(* Logix 5000 project; controller ACMI_PLC vendor 1 type 14 code 101 rev 19.11; software revision 19.01 *)
// Safety Rated PLC

TASK MainTask (periodic, rate 100 ms, priority 10, watchdog 2000 ms) : MainProgram
TASK SafetyTask (periodic, rate 20 ms, priority 2, watchdog 20 ms) : Main_Loop

MODULES
   Local : vendor 1 type 14 code 101 (1768Ctrl3Slot 0, Compact 0, rev 19.11)
      Temps : 1769-IR6 (Compact 1, rev 1.1, Input RPI 80 ms)
      SafetyEthernet : 1768-ENBT (1768 1, Ethernet 192.168.1.8, rev 4.4)
         PointIONet : 1734-AENT (Ethernet 192.168.1.9, rev 4.3, Output RPI 20 ms)
             : vendor 1 type 35 code 15 (PointIO 1, rev 2.1, Output RPI 20 ms, Input RPI 10 ms)
             : vendor 1 type 35 code 15 (PointIO 5, rev 2.1, Output RPI 20 ms, Input RPI 10 ms)
             : vendor 1 type 35 code 16 (PointIO 6, rev 2.1, Input RPI 10 ms, Output RPI 20 ms)
             : vendor 1 type 35 code 15 (PointIO 2, rev 2.1, Input RPI 10 ms, Output RPI 20 ms)
             : vendor 1 type 35 code 15 (PointIO 7, rev 2.1, Input RPI 10 ms, Output RPI 20 ms)
             : vendor 1 type 35 code 15 (PointIO 3, rev 2.1, Output RPI 20 ms, Input RPI 10 ms)
             : vendor 1 type 35 code 15 (PointIO 4, rev 2.1, Output RPI 20 ms, Input RPI 10 ms)
      PGRM : 1768-ENBT (1768 2, Ethernet 10.0.128.19, rev 4.1)
END_MODULES

TYPE BitStat :
STRUCT
   Hist : BOOL[4096];
   Top : INT;
   Sum : INT;
   Fault : BOOL;
END_STRUCT
END_TYPE

TYPE EVENT :
STRUCT
   TIME : TIME;
   EVENT : STRING;
END_STRUCT
END_TYPE

TYPE TIME :
STRUCT
   YEAR : DINT;
   MONTH : DINT;
   DAY : DINT;
   HOUR : DINT;
   MINUTE : DINT;
   SECOND : DINT;
   MICROSECOND : DINT;
END_STRUCT
END_TYPE

VAR_GLOBAL   (* controller tags *)
   A : DINT := 2047; {access Read Only}
   Abits : INT;
   ACMI_ADC_BITS : INT[2]; {access Read Only}
   ACMI_BEAM_DATA : REAL[7] := ([0] := 19.653, [1] := 16.0, [2] := -0.15, [5] := 82.0, [6] := 0.03); {access Read Only}
   ACMI_BEAM_Q : REAL := 19.653; {access Read Only}
   ACMI_BR_ACC : REAL; {access Read Only}
   ACMI_BR_CNT : DINT := 3278; {access Read Only}
   ACMI_BR_LIM : REAL := 82.0; {access Read Only}
   ACMI_CERTIFY : SINT; {access Read Only}
   ACMI_FAULT_CODE : DINT := 2097063; {access Read Only}
   ACMI_SHUTTER : BOOL; {access Read Only}
   ACMI_SR_LIM : REAL := 0.03; {access Read Only}
   ACMI_ST1_QAB : REAL := 19.021; {access Read Only}
   ACMI_ST1_QAB_AVG : REAL := 18.336615; {access Read Only}
   ACMI_ST1_QAB_HIST : DINT[31] := ([30] := 200); {access Read Only}
   ACMI_ST1_QAB_MAX : REAL := 19.713; {access Read Only}
   ACMI_ST1_QAB_MIN : REAL := -17.556; {access Read Only}
   ACMI_ST1_QAB_STD : REAL := 3362.0618; {access Read Only}
   ACMI_ST1_QBA : REAL := 19.152; {access Read Only}
   ACMI_ST1_QBA_AVG : REAL := 18.44839; {access Read Only}
   ACMI_ST1_QBA_HIST : DINT[31] := ([30] := 200); {access Read Only}
   ACMI_ST1_QBA_MAX : REAL := 19.713; {access Read Only}
   ACMI_ST1_QBA_MIN : REAL := -17.613; {access Read Only}
   ACMI_ST1_QBA_STD : REAL := 3396.1123; {access Read Only}
   ACMI_ST1_RST : SINT; {access Read Only}
   ACMI_ST2_QAB : REAL := 19.062; {access Read Only}
   ACMI_ST2_QAB_AVG : REAL := 18.345718; {access Read Only}
   ACMI_ST2_QAB_HIST : DINT[31] := ([30] := 200); {access Read Only}
   ACMI_ST2_QAB_MAX : REAL := 19.713; {access Read Only}
   ACMI_ST2_QAB_MIN : REAL := -17.572; {access Read Only}
   ACMI_ST2_QAB_STD : REAL := 3360.6584; {access Read Only}
   ACMI_ST2_QBA : REAL := 19.132; {access Read Only}
   ACMI_ST2_QBA_AVG : REAL := 18.451597; {access Read Only}
   ACMI_ST2_QBA_HIST : DINT[31] := ([30] := 200); {access Read Only}
   ACMI_ST2_QBA_MAX : REAL := 19.713; {access Read Only}
   ACMI_ST2_QBA_MIN : REAL := -17.638; {access Read Only}
   ACMI_ST2_QBA_STD : REAL := 3401.8562; {access Read Only}
   ACMI_ST2_RST : SINT; {access None}
   ACMI_ST_DATA : REAL[24] := ([0] := 19.021, [1] := 18.336615, [2] := 19.713, [3] := -17.556, [4] := 3362.0618, [5] := 19.152, [6] := 18.44839, [7] := 19.713, [8] := -17.613, [9] := 3396.1123, [10] := 0.75, [11] := 0.35, [12] := 19.062, [13] := 18.345718, [14] := 19.713, [15] := -17.572, [16] := 3360.6584, [17] := 19.132, [18] := 18.451597, [19] := 19.713, [20] := -17.638, [21] := 3401.8562, [22] := 16.4, [23] := 15.4); {access Read Only}
   ACMI_STAT_CODE : SINT; {access Read Only}
   ACMI_Stat_Size : INT := 200; {access Read Only}
   ACMI_TEMPS : INT[6] := ([0] := 210, [1] := 394, [2] := 256, [3] := 213, [4] := 172, [5] := 214); {access Read Only}
   ACMI_TIMING : SINT; {access Read Only}
   ACMI_TO_ACC : REAL; {access Read Only}
   ACMI_TO_CNT : DINT := 39; {access Read Only}
   ADCA : DINT := 2047; {access Read Only}
   ADCB : DINT := 58; {access Read Only}
   B : DINT := 58; {access Read Only}
   Bbits : INT;
   Beam_MaxQ : DINT := 16000; {constant, access Read Only}
   Beam_MinQ : DINT := -150; {constant, access Read Only}
   Beam_Q : DINT := 19653; {access Read Only}
   BR_Stack : DINT[7200]; {access Read Only}
   BR_Stack_MAX : DINT := 82000000; {constant, access Read Only}
   BR_Stack_Sum : DINT; {access Read Only}
   BR_Stack_Top : DINT := 923; {access Read Only}
   BSSS_CLOSED : ALIAS FOR PointIONet:7:I.Pt00Data;
   BYPASS_KEY : ALIAS FOR PointIONet:5:I.Pt07Data;
   FAULT_BEAM_BL : BOOL := 1; {access Read Only}
   FAULT_BEAM_HI : BOOL := 1; {access Read Only}
   FAULT_BEAM_LO : BOOL := 1;
   FAULT_BR_ACC : BOOL; {access Read Only}
   FAULT_CODE : DINT := 2097063;
   FAULT_QOW1 : BOOL := 1; {access Read Only}
   FAULT_QOW2 : BOOL; {access Read Only}
   FAULT_ST1_AB_HI : BOOL := 1; {access Read Only}
   FAULT_ST1_AB_LO : BOOL := 1; {access Read Only}
   FAULT_ST1_BA_HI : BOOL := 1; {access Read Only}
   FAULT_ST1_BA_LO : BOOL := 1; {access Read Only}
   FAULT_ST1_BLA : BOOL := 1; {access Read Only}
   FAULT_ST1_BLB : BOOL := 1; {access Read Only}
   FAULT_ST1_QAT : BOOL := 1; {access Read Only}
   FAULT_ST2_AB_HI : BOOL := 1; {access Read Only}
   FAULT_ST2_AB_LO : BOOL := 1; {access Read Only}
   FAULT_ST2_BA_HI : BOOL := 1; {access Read Only}
   FAULT_ST2_BA_LO : BOOL := 1; {access Read Only}
   FAULT_ST2_BLA : BOOL := 1; {access Read Only}
   FAULT_ST2_BLB : BOOL := 1; {access Read Only}
   FAULT_ST2_QAT : BOOL := 1; {access Read Only}
   FAULT_TO_ACC : BOOL; {access Read Only}
   FAULT_TWB : BOOL; {access Read Only}
   FAULT_WDT : BOOL; {access Read Only}
   HMI_BEAM_Q : REAL := 19.653; {access Read Only}
   HMI_Suppress : BOOL;
   Initialize : BOOL := 1; {access Read Only}
   LBSS_CLOSED : ALIAS FOR PointIONet:7:I.Pt01Data;
   PPS_RESET : ALIAS FOR PointIONet:7:I.Pt02Data;
   Q1AB : DINT;
   Relay_Error : BOOL; {access Read Only}
   RESET_ALL : ALIAS FOR PointIONet:5:I.Pt00Data;
   RESET_FAULT : ALIAS FOR PointIONet:5:I.Pt01Data;
   ST1_MaxQ : DINT := 750; {constant}
   ST1_MinQ : DINT := 350; {constant}
   ST1_QAB : DINT := 19021;
   ST1_QBA : DINT := 19152;
   ST1AB_Size : INT := 200;
   ST1BA_Size : INT := 200;
   ST2_MaxQ : DINT := 16400; {constant}
   ST2_MinQ : DINT := 15400; {constant}
   ST2_QAB : DINT := 19062;
   ST2_QBA : DINT := 19132;
   ST2AB_Size : INT := 200;
   ST2BA_Size : INT := 200;
   ST_HI_FAULT : BOOL := 1; {access Read Only}
   ST_LO_FAULT : BOOL; {access Read Only}
   ST_Size : BOOL := 1;
   ST_Type : BOOL;
   Stack_Size : DINT := 7067; {constant, access Read Only}
   TO_Cntr : COUNTER;
   TO_DISABLED : ALIAS FOR PointIONet:7:I.Pt03Data;
   TO_Stack : DINT[120]; {access Read Only}
   TO_Stack_MAX : DINT := 30000; {constant, access Read Only}
   TO_Stack_Size : DINT := 118; {constant, access Read Only}
   TO_Stack_Sum : DINT; {access Read Only}
   TO_Stack_Top : DINT := 47;
   TO_Status_Error : BOOL;
   Update_ST1_QAB : BOOL;
   Update_ST1_QBA : BOOL := 1;
   Update_ST2_QAB : BOOL := 1;
   Update_ST2_QBA : BOOL;
   Zero : DINT[7200]; {constant}
END_VAR

PROGRAM Event_Log   (* main routine Event_Log *)
VAR
   action_1 : BOOL; {access Read Only}
   action_10 : BOOL := 1; {access Read Only}
   action_11 : BOOL := 1;
   action_12 : BOOL;
   action_2 : BOOL := 1; {access Read Only}
   action_3 : BOOL; {access Read Only}
   action_4 : BOOL := 1; {access Read Only}
   action_5 : BOOL := 1; {access Read Only}
   action_6 : BOOL; {access Read Only}
   action_7 : BOOL := 1; {access Read Only}
   action_8 : BOOL; {access Read Only}
   action_9 : BOOL := 1; {access Read Only}
   Clear_Elog : BOOL := 1;
   Clock : TIME := (YEAR := 2025, MONTH := 4, DAY := 25, HOUR := 11, MINUTE := 37, SECOND := 34, MICROSECOND := 91157); {access Read Only}
   colon : STRING := ':'; {constant, access Read Only}
   Ehome : BOOL;
   Ehomeons : BOOL;
   Eindx : DINT;
   ELog : EVENT[1000] := ([0].TIME.YEAR := 2016, [0].TIME.MONTH := 6, [0].TIME.DAY := 14, [0].TIME.HOUR := 8, [0].TIME.MINUTE := 54, [0].TIME.SECOND := 13, [0].TIME.MICROSECOND := 99494, [0].EVENT := '2016/06/14   08:54:13   USER : RESET FAULT BUTTON PRESSED', [1].TIME.YEAR := 2016, [1].TIME.MONTH := 6, [1].TIME.DAY := 14, [1].TIME.HOUR := 15, [1].TIME.MINUTE := 7, [1].TIME.SECOND := 39, [1].TIME.MICROSECOND := 999465, [1].EVENT := '2016/06/14   15:07:39   FAULT : QOW1 : Charge Outside Window Detected', [2].TIME.YEAR := 2016, [2].TIME.MONTH := 6, [2].TIME.DAY := 14, [2].TIME.HOUR := 18, [2].TIME.MINUTE := 16, [2].TIME.SECOND := 9, [2].TIME.MICROSECOND := 400030, [2].EVENT := '2016/06/14   18:16:09   USER : PPS RESET FAULT BUTTON PRESSED', [3].TIME.YEAR := 2016, [3].TIME.MONTH := 6, [3].TIME.DAY := 14, [3].TIME.HOUR := 18, [3].TIME.MINUTE := 18, [3].TIME.SECOND := 25, [3].TIME.MICROSECOND := 799513, [3].EVENT := '2016/06/14   18:18:25   USER : PPS RESET FAULT BUTTON PRESSED', [4].TIME.YEAR := 2016, [4].TIME.MONTH := 6, [4].TIME.DAY := 14, [4].TIME.HOUR := 18, [4].TIME.MINUTE := 25, [4].TIME.SECOND := 9, [4].TIME.MICROSECOND := 99507, [4].EVENT := '2016/06/14   18:25:09   USER : PPS RESET FAULT BUTTON PRESSED', [5].TIME.YEAR := 2016, [5].TIME.MONTH := 6, [5].TIME.DAY := 14, [5].TIME.HOUR := 18, [5].TIME.MINUTE := 32, [5].TIME.SECOND := 13, [5].TIME.MICROSECOND := 899509, [5].EVENT := '2016/06/14   18:32:13   USER : PPS RESET FAULT BUTTON PRESSED', [6].TIME.YEAR := 2016, [6].TIME.MONTH := 6, [6].TIME.DAY := 14, [6].TIME.HOUR := 18, [6].TIME.MINUTE := 32, [6].TIME.SECOND := 14, [6].TIME.MICROSECOND := 399506, [6].EVENT := '2016/06/14   18:32:14   USER : PPS RESET FAULT BUTTON PRESSED', [7].TIME.YEAR := 2016, [7].TIME.MONTH := 6, [7].TIME.DAY := 14, [7].TIME.HOUR := 18,
        [7].TIME.MINUTE := 33, [7].TIME.SECOND := 34, [7].TIME.MICROSECOND := 499505, [7].EVENT := '2016/06/14   18:33:34   USER : PPS RESET FAULT BUTTON PRESSED', [8].TIME.YEAR := 2016, [8].TIME.MONTH := 6, [8].TIME.DAY := 14, [8].TIME.HOUR := 19, [8].TIME.MINUTE := 20, [8].TIME.SECOND := 22, [8].TIME.MICROSECOND := 599510, [8].EVENT := '2016/06/14   19:20:22   USER : PPS RESET FAULT BUTTON PRESSED', [9].TIME.YEAR := 2016, [9].TIME.MONTH := 6, [9].TIME.DAY := 14, [9].TIME.HOUR := 19, [9].TIME.MINUTE := 30, [9].TIME.SECOND := 2, [9].TIME.MICROSECOND := 699510, [9].EVENT := '2016/06/14   19:30:02   USER : PPS RESET FAULT BUTTON PRESSED', [10].TIME.YEAR := 2016, [10].TIME.MONTH := 6, [10].TIME.DAY := 14, [10].TIME.HOUR := 19, [10].TIME.MINUTE := 49, [10].TIME.SECOND := 34, [10].TIME.MICROSECOND := 999476, [10].EVENT := '2016/06/14   19:49:34   FAULT : QOW1 : Charge Outside Window Detected', [11].TIME.YEAR := 2016, [11].TIME.MONTH := 6, [11].TIME.DAY := 14, [11].TIME.HOUR := 19, [11].TIME.MINUTE := 50, [11].TIME.SECOND := 16, [11].TIME.MICROSECOND := 499512, [11].EVENT := '2016/06/14   19:50:16   USER : PPS RESET FAULT BUTTON PRESSED', [12].TIME.YEAR := 2016, [12].TIME.MONTH := 6, [12].TIME.DAY := 14, [12].TIME.HOUR := 19, [12].TIME.MINUTE := 50, [12].TIME.SECOND := 17, [12].TIME.MICROSECOND := 999514, [12].EVENT := '2016/06/14   19:50:17   USER : PPS RESET FAULT BUTTON PRESSED', [13].TIME.YEAR := 2016, [13].TIME.MONTH := 6, [13].TIME.DAY := 14, [13].TIME.HOUR := 19, [13].TIME.MINUTE := 58, [13].TIME.SECOND := 36, [13].TIME.MICROSECOND := 900080, [13].EVENT := '2016/06/14   19:58:36   USER : PPS RESET FAULT BUTTON PRESSED', [14].TIME.YEAR := 2016, [14].TIME.MONTH := 6, [14].TIME.DAY := 14, [14].TIME.HOUR := 21, [14].TIME.MINUTE := 23, [14].TIME.SECOND := 39, [14].TIME.MICROSECOND := 799512, [14].EVENT := '2016/06/14   21:23:39   USER : PPS RESET FAULT BUTTON PRESSED',
        [15].TIME.YEAR := 2016, [15].TIME.MONTH := 6, [15].TIME.DAY := 14, [15].TIME.HOUR := 22, [15].TIME.MINUTE := 11, [15].TIME.SECOND := 59, [15].TIME.MICROSECOND := 800029, [15].EVENT := '2016/06/14   22:11:59   USER : PPS RESET FAULT BUTTON PRESSED', [16].TIME.YEAR := 2016, [16].TIME.MONTH := 6, [16].TIME.DAY := 14, [16].TIME.HOUR := 23, [16].TIME.MINUTE := 1, [16].TIME.SECOND := 6, [16].TIME.MICROSECOND := 699515, [16].EVENT := '2016/06/14   23:01:06   USER : PPS RESET FAULT BUTTON PRESSED', [17].TIME.YEAR := 2016, [17].TIME.MONTH := 6, [17].TIME.DAY := 15, [17].TIME.MINUTE := 55, [17].TIME.SECOND := 57, [17].TIME.MICROSECOND := 899506, [17].EVENT := '2016/06/15   00:55:57   USER : PPS RESET FAULT BUTTON PRESSED', [18].TIME.YEAR := 2016, [18].TIME.MONTH := 6, [18].TIME.DAY := 15, [18].TIME.HOUR := 1, [18].TIME.MINUTE := 43, [18].TIME.SECOND := 11, [18].TIME.MICROSECOND := 799939, [18].EVENT := '2016/06/15   01:43:11   USER : PPS RESET FAULT BUTTON PRESSED', [19].TIME.YEAR := 2016, [19].TIME.MONTH := 6, [19].TIME.DAY := 15, [19].TIME.HOUR := 2, [19].TIME.MINUTE := 28, [19].TIME.SECOND := 20, [19].TIME.MICROSECOND := 599507, [19].EVENT := '2016/06/15   02:28:20   USER : PPS RESET FAULT BUTTON PRESSED', [20].TIME.YEAR := 2016, [20].TIME.MONTH := 6, [20].TIME.DAY := 15, [20].TIME.HOUR := 3, [20].TIME.MINUTE := 26, [20].TIME.SECOND := 38, [20].TIME.MICROSECOND := 999502, [20].EVENT := '2016/06/15   03:26:38   USER : PPS RESET FAULT BUTTON PRESSED', [21].TIME.YEAR := 2016, [21].TIME.MONTH := 6, [21].TIME.DAY := 15, [21].TIME.HOUR := 4, [21].TIME.MINUTE := 11, [21].TIME.SECOND := 32, [21].TIME.MICROSECOND := 999506, [21].EVENT := '2016/06/15   04:11:32   USER : PPS RESET FAULT BUTTON PRESSED', [22].TIME.YEAR := 2016, [22].TIME.MONTH := 6, [22].TIME.DAY := 15, [22].TIME.HOUR := 4, [22].TIME.MINUTE := 50,
        [22].TIME.SECOND := 6, [22].TIME.MICROSECOND := 899508, [22].EVENT := '2016/06/15   04:50:06   USER : PPS RESET FAULT BUTTON PRESSED', [23].TIME.YEAR := 2016, [23].TIME.MONTH := 6, [23].TIME.DAY := 15, [23].TIME.HOUR := 5, [23].TIME.MINUTE := 8, [23].TIME.SECOND := 40, [23].TIME.MICROSECOND := 199505, [23].EVENT := '2016/06/15   05:08:40   USER : PPS RESET FAULT BUTTON PRESSED', [24].TIME.YEAR := 2016, [24].TIME.MONTH := 6, [24].TIME.DAY := 15, [24].TIME.HOUR := 5, [24].TIME.MINUTE := 36, [24].TIME.SECOND := 52, [24].TIME.MICROSECOND := 99507, [24].EVENT := '2016/06/15   05:36:52   USER : PPS RESET FAULT BUTTON PRESSED', [25].TIME.YEAR := 2016, [25].TIME.MONTH := 6, [25].TIME.DAY := 15, [25].TIME.HOUR := 7, [25].TIME.MINUTE := 29, [25].TIME.SECOND := 5, [25].TIME.MICROSECOND := 499507, [25].EVENT := '2016/06/15   07:29:05   USER : PPS RESET FAULT BUTTON PRESSED', [26].TIME.YEAR := 2016, [26].TIME.MONTH := 6, [26].TIME.DAY := 15, [26].TIME.HOUR := 9, [26].TIME.MINUTE := 57, [26].TIME.SECOND := 54, [26].TIME.MICROSECOND := 799464, [26].EVENT := '2016/06/15   09:57:54   FAULT : QOW1 : Charge Outside Window Detected', [27].TIME.YEAR := 2016, [27].TIME.MONTH := 6, [27].TIME.DAY := 15, [27].TIME.HOUR := 12, [27].TIME.MINUTE := 48, [27].TIME.SECOND := 48, [27].TIME.MICROSECOND := 999725, [27].EVENT := '2016/06/15   12:48:48   USER : PPS RESET FAULT BUTTON PRESSED', [28].TIME.YEAR := 2016, [28].TIME.MONTH := 6, [28].TIME.DAY := 15, [28].TIME.HOUR := 16, [28].TIME.MINUTE := 54, [28].TIME.SECOND := 28, [28].TIME.MICROSECOND := 299521, [28].EVENT := '2016/06/15   16:54:28   USER : PPS RESET FAULT BUTTON PRESSED', [29].TIME.YEAR := 2016, [29].TIME.MONTH := 6, [29].TIME.DAY := 15, [29].TIME.HOUR := 17, [29].TIME.MINUTE := 29, [29].TIME.SECOND := 30, [29].TIME.MICROSECOND := 299467, [29].EVENT := '2016/06/15   17:29:30   FAULT : QOW1 : Charge Outside Window Detected', [30].TIME.YEAR := 2016,
        [30].TIME.MONTH := 6, [30].TIME.DAY := 15, [30].TIME.HOUR := 17, [30].TIME.MINUTE := 30, [30].TIME.MICROSECOND := 600025, [30].EVENT := '2016/06/15   17:30:00   USER : PPS RESET FAULT BUTTON PRESSED', [31].TIME.YEAR := 2016, [31].TIME.MONTH := 6, [31].TIME.DAY := 15, [31].TIME.HOUR := 17, [31].TIME.MINUTE := 30, [31].TIME.SECOND := 48, [31].TIME.MICROSECOND := 99559, [31].EVENT := '2016/06/15   17:30:48   USER : PPS RESET FAULT BUTTON PRESSED', [32].TIME.YEAR := 2016, [32].TIME.MONTH := 6, [32].TIME.DAY := 15, [32].TIME.HOUR := 17, [32].TIME.MINUTE := 31, [32].TIME.SECOND := 16, [32].TIME.MICROSECOND := 999943, [32].EVENT := '2016/06/15   17:31:16   USER : PPS RESET FAULT BUTTON PRESSED', [33].TIME.YEAR := 2016, [33].TIME.MONTH := 6, [33].TIME.DAY := 15, [33].TIME.HOUR := 17, [33].TIME.MINUTE := 31, [33].TIME.SECOND := 20, [33].TIME.MICROSECOND := 699565, [33].EVENT := '2016/06/15   17:31:20   USER : PPS RESET FAULT BUTTON PRESSED', [34].TIME.YEAR := 2016, [34].TIME.MONTH := 6, [34].TIME.DAY := 15, [34].TIME.HOUR := 17, [34].TIME.MINUTE := 33, [34].TIME.SECOND := 7, [34].TIME.MICROSECOND := 599508, [34].EVENT := '2016/06/15   17:33:07   USER : PPS RESET FAULT BUTTON PRESSED', [35].TIME.YEAR := 2016, [35].TIME.MONTH := 6, [35].TIME.DAY := 15, [35].TIME.HOUR := 17, [35].TIME.MINUTE := 37, [35].TIME.SECOND := 31, [35].TIME.MICROSECOND := 400126, [35].EVENT := '2016/06/15   17:37:31   USER : PPS RESET FAULT BUTTON PRESSED', [36].TIME.YEAR := 2016, [36].TIME.MONTH := 6, [36].TIME.DAY := 15, [36].TIME.HOUR := 17, [36].TIME.MINUTE := 37, [36].TIME.SECOND := 35, [36].TIME.MICROSECOND := 18, [36].EVENT := '2016/06/15   17:37:35   USER : PPS RESET FAULT BUTTON PRESSED', [37].TIME.YEAR := 2016, [37].TIME.MONTH := 6, [37].TIME.DAY := 15, [37].TIME.HOUR := 22, [37].TIME.MINUTE := 8, [37].TIME.SECOND := 46,
        [37].TIME.MICROSECOND := 799505, [37].EVENT := '2016/06/15   22:08:46   USER : PPS RESET FAULT BUTTON PRESSED', [38].TIME.YEAR := 2016, [38].TIME.MONTH := 6, [38].TIME.DAY := 15, [38].TIME.HOUR := 22, [38].TIME.MINUTE := 26, [38].TIME.SECOND := 18, [38].TIME.MICROSECOND := 799507, [38].EVENT := '2016/06/15   22:26:18   USER : PPS RESET FAULT BUTTON PRESSED', [39].TIME.YEAR := 2016, [39].TIME.MONTH := 6, [39].TIME.DAY := 15, [39].TIME.HOUR := 22, [39].TIME.MINUTE := 26, [39].TIME.SECOND := 19, [39].TIME.MICROSECOND := 999507, [39].EVENT := '2016/06/15   22:26:19   USER : PPS RESET FAULT BUTTON PRESSED', [40].TIME.YEAR := 2016, [40].TIME.MONTH := 6, [40].TIME.DAY := 16, [40].TIME.HOUR := 5, [40].TIME.MINUTE := 59, [40].TIME.SECOND := 17, [40].TIME.MICROSECOND := 599513, [40].EVENT := '2016/06/16   05:59:17   USER : PPS RESET FAULT BUTTON PRESSED', [41].TIME.YEAR := 2016, [41].TIME.MONTH := 6, [41].TIME.DAY := 16, [41].TIME.HOUR := 7, [41].TIME.MINUTE := 7, [41].TIME.SECOND := 40, [41].TIME.MICROSECOND := 699942, [41].EVENT := '2016/06/16   07:07:40   USER : PPS RESET FAULT BUTTON PRESSED', [42].TIME.YEAR := 2016, [42].TIME.MONTH := 6, [42].TIME.DAY := 16, [42].TIME.HOUR := 7, [42].TIME.MINUTE := 30, [42].TIME.SECOND := 30, [42].TIME.MICROSECOND := 299509, [42].EVENT := '2016/06/16   07:30:30   USER : PPS RESET FAULT BUTTON PRESSED', [43].TIME.YEAR := 2016, [43].TIME.MONTH := 6, [43].TIME.DAY := 16, [43].TIME.HOUR := 7, [43].TIME.MINUTE := 37, [43].TIME.SECOND := 3, [43].TIME.MICROSECOND := 999505, [43].EVENT := '2016/06/16   07:37:03   USER : PPS RESET FAULT BUTTON PRESSED', [44].TIME.YEAR := 2016, [44].TIME.MONTH := 6, [44].TIME.DAY := 17, [44].TIME.HOUR := 3, [44].TIME.MINUTE := 10, [44].TIME.SECOND := 56, [44].TIME.MICROSECOND := 399504, [44].EVENT := '2016/06/17   03:10:56   USER : PPS RESET FAULT BUTTON PRESSED', [45].TIME.YEAR := 2016, [45].TIME.MONTH := 6,
        [45].TIME.DAY := 17, [45].TIME.HOUR := 3, [45].TIME.MINUTE := 10, [45].TIME.SECOND := 56, [45].TIME.MICROSECOND := 999667, [45].EVENT := '2016/06/17   03:10:56   USER : PPS RESET FAULT BUTTON PRESSED', [46].TIME.YEAR := 2016, [46].TIME.MONTH := 6, [46].TIME.DAY := 19, [46].TIME.HOUR := 6, [46].TIME.MINUTE := 3, [46].TIME.SECOND := 57, [46].TIME.MICROSECOND := 499514, [46].EVENT := '2016/06/19   06:03:57   USER : PPS RESET FAULT BUTTON PRESSED', [47].TIME.YEAR := 2016, [47].TIME.MONTH := 6, [47].TIME.DAY := 19, [47].TIME.HOUR := 6, [47].TIME.MINUTE := 16, [47].TIME.SECOND := 38, [47].TIME.MICROSECOND := 199508, [47].EVENT := '2016/06/19   06:16:38   USER : PPS RESET FAULT BUTTON PRESSED', [48].TIME.YEAR := 2016, [48].TIME.MONTH := 6, [48].TIME.DAY := 19, [48].TIME.HOUR := 11, [48].TIME.MINUTE := 46, [48].TIME.SECOND := 51, [48].TIME.MICROSECOND := 499501, [48].EVENT := '2016/06/19   11:46:51   USER : PPS RESET FAULT BUTTON PRESSED', [49].TIME.YEAR := 2016, [49].TIME.MONTH := 6, [49].TIME.DAY := 19, [49].TIME.HOUR := 11, [49].TIME.MINUTE := 46, [49].TIME.SECOND := 54, [49].TIME.MICROSECOND := 899719, [49].EVENT := '2016/06/19   11:46:54   USER : PPS RESET FAULT BUTTON PRESSED', [50].TIME.YEAR := 2016, [50].TIME.MONTH := 6, [50].TIME.DAY := 19, [50].TIME.HOUR := 11, [50].TIME.MINUTE := 47, [50].TIME.MICROSECOND := 99505, [50].EVENT := '2016/06/19   11:47:00   USER : PPS RESET FAULT BUTTON PRESSED', [51].TIME.YEAR := 2016, [51].TIME.MONTH := 6, [51].TIME.DAY := 19, [51].TIME.HOUR := 12, [51].TIME.MINUTE := 28, [51].TIME.SECOND := 56, [51].TIME.MICROSECOND := 799506, [51].EVENT := '2016/06/19   12:28:56   USER : PPS RESET FAULT BUTTON PRESSED', [52].TIME.YEAR := 2016, [52].TIME.MONTH := 6, [52].TIME.DAY := 19, [52].TIME.HOUR := 12, [52].TIME.MINUTE := 29, [52].TIME.SECOND := 10, [52].TIME.MICROSECOND := 299944,
        [52].EVENT := '2016/06/19   12:29:10   USER : PPS RESET FAULT BUTTON PRESSED', [53].TIME.YEAR := 2016, [53].TIME.MONTH := 6, [53].TIME.DAY := 20, [53].TIME.HOUR := 2, [53].TIME.MINUTE := 56, [53].TIME.SECOND := 49, [53].TIME.MICROSECOND := 799466, [53].EVENT := '2016/06/20   02:56:49   FAULT : QOW1 : Charge Outside Window Detected', [54].TIME.YEAR := 2016, [54].TIME.MONTH := 6, [54].TIME.DAY := 20, [54].TIME.HOUR := 3, [54].TIME.MINUTE := 1, [54].TIME.SECOND := 12, [54].TIME.MICROSECOND := 899513, [54].EVENT := '2016/06/20   03:01:12   USER : PPS RESET FAULT BUTTON PRESSED', [55].TIME.YEAR := 2016, [55].TIME.MONTH := 6, [55].TIME.DAY := 20, [55].TIME.HOUR := 9, [55].TIME.MINUTE := 53, [55].TIME.SECOND := 57, [55].TIME.MICROSECOND := 599892, [55].EVENT := '2016/06/20   09:53:57   FAULT : QOW1 : Charge Outside Window Detected', [56].TIME.YEAR := 2016, [56].TIME.MONTH := 6, [56].TIME.DAY := 20, [56].TIME.HOUR := 9, [56].TIME.MINUTE := 56, [56].TIME.SECOND := 28, [56].TIME.MICROSECOND := 999507, [56].EVENT := '2016/06/20   09:56:28   USER : PPS RESET FAULT BUTTON PRESSED', [57].TIME.YEAR := 2016, [57].TIME.MONTH := 6, [57].TIME.DAY := 20, [57].TIME.HOUR := 9, [57].TIME.MINUTE := 57, [57].TIME.MICROSECOND := 399561, [57].EVENT := '2016/06/20   09:57:00   USER : PPS RESET FAULT BUTTON PRESSED', [58].TIME.YEAR := 2016, [58].TIME.MONTH := 6, [58].TIME.DAY := 20, [58].TIME.HOUR := 11, [58].TIME.MINUTE := 53, [58].TIME.SECOND := 14, [58].TIME.MICROSECOND := 199466, [58].EVENT := '2016/06/20   11:53:14   FAULT : QOW1 : Charge Outside Window Detected', [59].TIME.YEAR := 2016, [59].TIME.MONTH := 6, [59].TIME.DAY := 20, [59].TIME.HOUR := 12, [59].TIME.MINUTE := 17, [59].TIME.SECOND := 3, [59].TIME.MICROSECOND := 999504, [59].EVENT := '2016/06/20   12:17:03   USER : PPS RESET FAULT BUTTON PRESSED', [60].TIME.YEAR := 2016, [60].TIME.MONTH := 6, [60].TIME.DAY := 20, [60].TIME.HOUR := 12,
        [60].TIME.MINUTE := 19, [60].TIME.SECOND := 21, [60].TIME.MICROSECOND := 699508, [60].EVENT := '2016/06/20   12:19:21   USER : PPS RESET FAULT BUTTON PRESSED', [61].TIME.YEAR := 2016, [61].TIME.MONTH := 6, [61].TIME.DAY := 20, [61].TIME.HOUR := 15, [61].TIME.MINUTE := 7, [61].TIME.SECOND := 52, [61].TIME.MICROSECOND := 999508, [61].EVENT := '2016/06/20   15:07:52   USER : PPS RESET FAULT BUTTON PRESSED', [62].TIME.YEAR := 2016, [62].TIME.MONTH := 6, [62].TIME.DAY := 20, [62].TIME.HOUR := 15, [62].TIME.MINUTE := 8, [62].TIME.MICROSECOND := 500039, [62].EVENT := '2016/06/20   15:08:00   USER : PPS RESET FAULT BUTTON PRESSED', [63].TIME.YEAR := 2016, [63].TIME.MONTH := 6, [63].TIME.DAY := 21, [63].TIME.HOUR := 6, [63].TIME.MINUTE := 34, [63].TIME.SECOND := 32, [63].TIME.MICROSECOND := 799508, [63].EVENT := '2016/06/21   06:34:32   USER : PPS RESET FAULT BUTTON PRESSED', [64].TIME.YEAR := 2016, [64].TIME.MONTH := 6, [64].TIME.DAY := 21, [64].TIME.HOUR := 16, [64].TIME.MINUTE := 11, [64].TIME.SECOND := 44, [64].TIME.MICROSECOND := 699508, [64].EVENT := '2016/06/21   16:11:44   USER : PPS RESET FAULT BUTTON PRESSED', [65].TIME.YEAR := 2016, [65].TIME.MONTH := 6, [65].TIME.DAY := 22, [65].TIME.HOUR := 10, [65].TIME.MINUTE := 49, [65].TIME.SECOND := 42, [65].TIME.MICROSECOND := 899505, [65].EVENT := '2016/06/22   10:49:42   USER : PPS RESET FAULT BUTTON PRESSED', [66].TIME.YEAR := 2016, [66].TIME.MONTH := 6, [66].TIME.DAY := 23, [66].TIME.HOUR := 10, [66].TIME.MINUTE := 34, [66].TIME.SECOND := 24, [66].TIME.MICROSECOND := 99613, [66].EVENT := '2016/06/23   10:34:24   FAULT : QOW1 : Charge Outside Window Detected', [67].TIME.YEAR := 2016, [67].TIME.MONTH := 6, [67].TIME.DAY := 23, [67].TIME.HOUR := 10, [67].TIME.MINUTE := 34, [67].TIME.SECOND := 59, [67].TIME.MICROSECOND := 699586, [67].EVENT := '2016/06/23   10:34:59   USER : PPS RESET FAULT BUTTON PRESSED', [68].TIME.YEAR := 2016,
        [68].TIME.MONTH := 6, [68].TIME.DAY := 23, [68].TIME.HOUR := 10, [68].TIME.MINUTE := 35, [68].TIME.SECOND := 3, [68].TIME.MICROSECOND := 499555, [68].EVENT := '2016/06/23   10:35:03   USER : PPS RESET FAULT BUTTON PRESSED', [69].TIME.YEAR := 2016, [69].TIME.MONTH := 6, [69].TIME.DAY := 23, [69].TIME.HOUR := 10, [69].TIME.MINUTE := 35, [69].TIME.SECOND := 6, [69].TIME.MICROSECOND := 999613, [69].EVENT := '2016/06/23   10:35:06   USER : PPS RESET FAULT BUTTON PRESSED', [70].TIME.YEAR := 2016, [70].TIME.MONTH := 6, [70].TIME.DAY := 23, [70].TIME.HOUR := 13, [70].TIME.MINUTE := 40, [70].TIME.SECOND := 28, [70].TIME.MICROSECOND := 199506, [70].EVENT := '2016/06/23   13:40:28   USER : PPS RESET FAULT BUTTON PRESSED', [71].TIME.YEAR := 2016, [71].TIME.MONTH := 6, [71].TIME.DAY := 23, [71].TIME.HOUR := 19, [71].TIME.MINUTE := 19, [71].TIME.SECOND := 36, [71].TIME.MICROSECOND := 99466, [71].EVENT := '2016/06/23   19:19:36   FAULT : QOW1 : Charge Outside Window Detected', [72].TIME.YEAR := 2016, [72].TIME.MONTH := 6, [72].TIME.DAY := 23, [72].TIME.HOUR := 19, [72].TIME.MINUTE := 21, [72].TIME.SECOND := 43, [72].TIME.MICROSECOND := 799507, [72].EVENT := '2016/06/23   19:21:43   USER : PPS RESET FAULT BUTTON PRESSED', [73].TIME.YEAR := 2016, [73].TIME.MONTH := 6, [73].TIME.DAY := 23, [73].TIME.HOUR := 19, [73].TIME.MINUTE := 21, [73].TIME.SECOND := 47, [73].TIME.MICROSECOND := 899509, [73].EVENT := '2016/06/23   19:21:47   USER : PPS RESET FAULT BUTTON PRESSED', [74].TIME.YEAR := 2016, [74].TIME.MONTH := 6, [74].TIME.DAY := 24, [74].TIME.HOUR := 14, [74].TIME.MINUTE := 11, [74].TIME.SECOND := 36, [74].TIME.MICROSECOND := 299508, [74].EVENT := '2016/06/24   14:11:36   USER : PPS RESET FAULT BUTTON PRESSED', [75].TIME.YEAR := 2016, [75].TIME.MONTH := 6, [75].TIME.DAY := 24, [75].TIME.HOUR := 14, [75].TIME.MINUTE := 12,
        [75].TIME.SECOND := 11, [75].TIME.MICROSECOND := 399510, [75].EVENT := '2016/06/24   14:12:11   USER : PPS RESET FAULT BUTTON PRESSED', [76].TIME.YEAR := 2016, [76].TIME.MONTH := 6, [76].TIME.DAY := 24, [76].TIME.HOUR := 19, [76].TIME.MINUTE := 38, [76].TIME.SECOND := 16, [76].TIME.MICROSECOND := 899505, [76].EVENT := '2016/06/24   19:38:16   USER : PPS RESET FAULT BUTTON PRESSED', [77].TIME.YEAR := 2016, [77].TIME.MONTH := 6, [77].TIME.DAY := 24, [77].TIME.HOUR := 19, [77].TIME.MINUTE := 38, [77].TIME.SECOND := 17, [77].TIME.MICROSECOND := 299513, [77].EVENT := '2016/06/24   19:38:17   USER : PPS RESET FAULT BUTTON PRESSED', [78].TIME.YEAR := 2016, [78].TIME.MONTH := 6, [78].TIME.DAY := 26, [78].TIME.HOUR := 7, [78].TIME.MINUTE := 52, [78].TIME.SECOND := 23, [78].TIME.MICROSECOND := 200116, [78].EVENT := '2016/06/26   07:52:23   FAULT : QOW1 : Charge Outside Window Detected', [79].TIME.YEAR := 2016, [79].TIME.MONTH := 6, [79].TIME.DAY := 26, [79].TIME.HOUR := 10, [79].TIME.MINUTE := 40, [79].TIME.SECOND := 12, [79].TIME.MICROSECOND := 799507, [79].EVENT := '2016/06/26   10:40:12   USER : PPS RESET FAULT BUTTON PRESSED', [80].TIME.YEAR := 2016, [80].TIME.MONTH := 6, [80].TIME.DAY := 26, [80].TIME.HOUR := 10, [80].TIME.MINUTE := 40, [80].TIME.SECOND := 42, [80].TIME.MICROSECOND := 900026, [80].EVENT := '2016/06/26   10:40:42   USER : PPS RESET FAULT BUTTON PRESSED', [81].TIME.YEAR := 2016, [81].TIME.MONTH := 6, [81].TIME.DAY := 26, [81].TIME.HOUR := 12, [81].TIME.MINUTE := 6, [81].TIME.SECOND := 57, [81].TIME.MICROSECOND := 399947, [81].EVENT := '2016/06/26   12:06:57   USER : PPS RESET FAULT BUTTON PRESSED', [82].TIME.YEAR := 2016, [82].TIME.MONTH := 6, [82].TIME.DAY := 26, [82].TIME.HOUR := 15, [82].TIME.MINUTE := 33, [82].TIME.SECOND := 30, [82].TIME.MICROSECOND := 599505, [82].EVENT := '2016/06/26   15:33:30   USER : PPS RESET FAULT BUTTON PRESSED', [83].TIME.YEAR := 2016,
        [83].TIME.MONTH := 6, [83].TIME.DAY := 26, [83].TIME.HOUR := 15, [83].TIME.MINUTE := 33, [83].TIME.SECOND := 41, [83].TIME.MICROSECOND := 599505, [83].EVENT := '2016/06/26   15:33:41   USER : PPS RESET FAULT BUTTON PRESSED', [84].TIME.YEAR := 2016, [84].TIME.MONTH := 6, [84].TIME.DAY := 26, [84].TIME.HOUR := 15, [84].TIME.MINUTE := 33, [84].TIME.SECOND := 50, [84].TIME.MICROSECOND := 199507, [84].EVENT := '2016/06/26   15:33:50   USER : PPS RESET FAULT BUTTON PRESSED', [85].TIME.YEAR := 2016, [85].TIME.MONTH := 6, [85].TIME.DAY := 26, [85].TIME.HOUR := 15, [85].TIME.MINUTE := 33, [85].TIME.SECOND := 53, [85].TIME.MICROSECOND := 299726, [85].EVENT := '2016/06/26   15:33:53   USER : PPS RESET FAULT BUTTON PRESSED', [86].TIME.YEAR := 2016, [86].TIME.MONTH := 6, [86].TIME.DAY := 26, [86].TIME.HOUR := 15, [86].TIME.MINUTE := 34, [86].TIME.MICROSECOND := 700024, [86].EVENT := '2016/06/26   15:34:00   USER : PPS RESET FAULT BUTTON PRESSED', [87].TIME.YEAR := 2016, [87].TIME.MONTH := 6, [87].TIME.DAY := 26, [87].TIME.HOUR := 15, [87].TIME.MINUTE := 34, [87].TIME.SECOND := 58, [87].TIME.MICROSECOND := 499513, [87].EVENT := '2016/06/26   15:34:58   USER : PPS RESET FAULT BUTTON PRESSED', [88].TIME.YEAR := 2016, [88].TIME.MONTH := 6, [88].TIME.DAY := 26, [88].TIME.HOUR := 15, [88].TIME.MINUTE := 46, [88].TIME.SECOND := 2, [88].TIME.MICROSECOND := 799503, [88].EVENT := '2016/06/26   15:46:02   USER : PPS RESET FAULT BUTTON PRESSED', [89].TIME.YEAR := 2016, [89].TIME.MONTH := 6, [89].TIME.DAY := 26, [89].TIME.HOUR := 16, [89].TIME.MINUTE := 36, [89].TIME.SECOND := 3, [89].TIME.MICROSECOND := 99521, [89].EVENT := '2016/06/26   16:36:03   USER : PPS RESET FAULT BUTTON PRESSED', [90].TIME.YEAR := 2016, [90].TIME.MONTH := 6, [90].TIME.DAY := 26, [90].TIME.HOUR := 16, [90].TIME.MINUTE := 36, [90].TIME.SECOND := 5,
        [90].TIME.MICROSECOND := 299935, [90].EVENT := '2016/06/26   16:36:05   USER : PPS RESET FAULT BUTTON PRESSED', [91].TIME.YEAR := 2016, [91].TIME.MONTH := 6, [91].TIME.DAY := 26, [91].TIME.HOUR := 16, [91].TIME.MINUTE := 39, [91].TIME.SECOND := 8, [91].TIME.MICROSECOND := 99510, [91].EVENT := '2016/06/26   16:39:08   USER : PPS RESET FAULT BUTTON PRESSED', [92].TIME.YEAR := 2016, [92].TIME.MONTH := 6, [92].TIME.DAY := 26, [92].TIME.HOUR := 16, [92].TIME.MINUTE := 53, [92].TIME.SECOND := 12, [92].TIME.MICROSECOND := 299942, [92].EVENT := '2016/06/26   16:53:12   USER : PPS RESET FAULT BUTTON PRESSED', [93].TIME.YEAR := 2016, [93].TIME.MONTH := 6, [93].TIME.DAY := 27, [93].TIME.HOUR := 8, [93].TIME.MINUTE := 50, [93].TIME.SECOND := 16, [93].TIME.MICROSECOND := 33, [93].EVENT := '2016/06/27   08:50:16   USER : PPS RESET FAULT BUTTON PRESSED', [94].TIME.YEAR := 2016, [94].TIME.MONTH := 6, [94].TIME.DAY := 27, [94].TIME.HOUR := 11, [94].TIME.MINUTE := 25, [94].TIME.SECOND := 14, [94].TIME.MICROSECOND := 99562, [94].EVENT := '2016/06/27   11:25:14   USER : PPS RESET FAULT BUTTON PRESSED', [95].TIME.YEAR := 2016, [95].TIME.MONTH := 6, [95].TIME.DAY := 27, [95].TIME.HOUR := 11, [95].TIME.MINUTE := 46, [95].TIME.SECOND := 8, [95].TIME.MICROSECOND := 799509, [95].EVENT := '2016/06/27   11:46:08   USER : PPS RESET FAULT BUTTON PRESSED', [96].TIME.YEAR := 2016, [96].TIME.MONTH := 6, [96].TIME.DAY := 27, [96].TIME.HOUR := 14, [96].TIME.MINUTE := 38, [96].TIME.SECOND := 8, [96].TIME.MICROSECOND := 899507, [96].EVENT := '2016/06/27   14:38:08   USER : PPS RESET FAULT BUTTON PRESSED', [97].TIME.YEAR := 2016, [97].TIME.MONTH := 6, [97].TIME.DAY := 27, [97].TIME.HOUR := 14, [97].TIME.MINUTE := 38, [97].TIME.SECOND := 13, [97].TIME.MICROSECOND := 799511, [97].EVENT := '2016/06/27   14:38:13   USER : PPS RESET FAULT BUTTON PRESSED', [98].TIME.YEAR := 2016, [98].TIME.MONTH := 6,
        [98].TIME.DAY := 27, [98].TIME.HOUR := 14, [98].TIME.MINUTE := 39, [98].TIME.SECOND := 25, [98].TIME.MICROSECOND := 199509, [98].EVENT := '2016/06/27   14:39:25   USER : PPS RESET FAULT BUTTON PRESSED', [99].TIME.YEAR := 2016, [99].TIME.MONTH := 6, [99].TIME.DAY := 27, [99].TIME.HOUR := 14, [99].TIME.MINUTE := 41, [99].TIME.SECOND := 11, [99].TIME.MICROSECOND := 499511, [99].EVENT := '2016/06/27   14:41:11   USER : PPS RESET FAULT BUTTON PRESSED', [100].TIME.YEAR := 2016, [100].TIME.MONTH := 6, [100].TIME.DAY := 27, [100].TIME.HOUR := 19, [100].TIME.MINUTE := 42, [100].TIME.SECOND := 41, [100].TIME.MICROSECOND := 999515, [100].EVENT := '2016/06/27   19:42:41   USER : PPS RESET FAULT BUTTON PRESSED', [101].TIME.YEAR := 2016, [101].TIME.MONTH := 6, [101].TIME.DAY := 27, [101].TIME.HOUR := 19, [101].TIME.MINUTE := 42, [101].TIME.SECOND := 56, [101].TIME.MICROSECOND := 899473, [101].EVENT := '2016/06/27   19:42:56   FAULT : QOW1 : Charge Outside Window Detected', [102].TIME.YEAR := 2016, [102].TIME.MONTH := 6, [102].TIME.DAY := 27, [102].TIME.HOUR := 19, [102].TIME.MINUTE := 43, [102].TIME.SECOND := 6, [102].TIME.MICROSECOND := 99514, [102].EVENT := '2016/06/27   19:43:06   USER : PPS RESET FAULT BUTTON PRESSED', [103].TIME.YEAR := 2016, [103].TIME.MONTH := 6, [103].TIME.DAY := 28, [103].TIME.HOUR := 8, [103].TIME.MINUTE := 48, [103].TIME.MICROSECOND := 899470, [103].EVENT := '2016/06/28   08:48:00   FAULT : QOW1 : Charge Outside Window Detected', [104].TIME.YEAR := 2016, [104].TIME.MONTH := 6, [104].TIME.DAY := 28, [104].TIME.HOUR := 23, [104].TIME.MINUTE := 28, [104].TIME.SECOND := 39, [104].TIME.MICROSECOND := 399496, [104].EVENT := '2016/06/28   23:28:39   USER : RESET FAULT BUTTON PRESSED', [105].TIME.YEAR := 2016, [105].TIME.MONTH := 6, [105].TIME.DAY := 28, [105].TIME.HOUR := 23, [105].TIME.MINUTE := 28, [105].TIME.SECOND := 41, [105].TIME.MICROSECOND := 999490,
        [105].EVENT := '2016/06/28   23:28:41   USER : RESET FAULT BUTTON PRESSED', [106].TIME.YEAR := 2016, [106].TIME.MONTH := 6, [106].TIME.DAY := 29, [106].TIME.HOUR := 9, [106].TIME.MINUTE := 25, [106].TIME.SECOND := 28, [106].TIME.MICROSECOND := 899510, [106].EVENT := '2016/06/29   09:25:28   USER : PPS RESET FAULT BUTTON PRESSED', [107].TIME.YEAR := 2016, [107].TIME.MONTH := 6, [107].TIME.DAY := 29, [107].TIME.HOUR := 9, [107].TIME.MINUTE := 26, [107].TIME.SECOND := 43, [107].TIME.MICROSECOND := 499506, [107].EVENT := '2016/06/29   09:26:43   USER : PPS RESET FAULT BUTTON PRESSED', [108].TIME.YEAR := 2016, [108].TIME.MONTH := 6, [108].TIME.DAY := 29, [108].TIME.HOUR := 9, [108].TIME.MINUTE := 37, [108].TIME.SECOND := 5, [108].TIME.MICROSECOND := 699512, [108].EVENT := '2016/06/29   09:37:05   USER : PPS RESET FAULT BUTTON PRESSED', [109].TIME.YEAR := 2016, [109].TIME.MONTH := 6, [109].TIME.DAY := 29, [109].TIME.HOUR := 9, [109].TIME.MINUTE := 45, [109].TIME.SECOND := 12, [109].TIME.MICROSECOND := 299508, [109].EVENT := '2016/06/29   09:45:12   USER : PPS RESET FAULT BUTTON PRESSED', [110].TIME.YEAR := 2016, [110].TIME.MONTH := 6, [110].TIME.DAY := 29, [110].TIME.HOUR := 9, [110].TIME.MINUTE := 45, [110].TIME.SECOND := 18, [110].TIME.MICROSECOND := 99508, [110].EVENT := '2016/06/29   09:45:18   USER : PPS RESET FAULT BUTTON PRESSED', [111].TIME.YEAR := 2016, [111].TIME.MONTH := 6, [111].TIME.DAY := 29, [111].TIME.HOUR := 9, [111].TIME.MINUTE := 47, [111].TIME.SECOND := 38, [111].TIME.MICROSECOND := 999504, [111].EVENT := '2016/06/29   09:47:38   USER : PPS RESET FAULT BUTTON PRESSED', [112].TIME.YEAR := 2016, [112].TIME.MONTH := 6, [112].TIME.DAY := 29, [112].TIME.HOUR := 9, [112].TIME.MINUTE := 50, [112].TIME.SECOND := 52, [112].TIME.MICROSECOND := 499511, [112].EVENT := '2016/06/29   09:50:52   USER : PPS RESET FAULT BUTTON PRESSED', [113].TIME.YEAR := 2016, [113].TIME.MONTH := 6, [113].TIME.DAY := 29,
        [113].TIME.HOUR := 9, [113].TIME.MINUTE := 52, [113].TIME.SECOND := 15, [113].TIME.MICROSECOND := 699648, [113].EVENT := '2016/06/29   09:52:15   USER : PPS RESET FAULT BUTTON PRESSED', [114].TIME.YEAR := 2016, [114].TIME.MONTH := 6, [114].TIME.DAY := 29, [114].TIME.HOUR := 9, [114].TIME.MINUTE := 53, [114].TIME.SECOND := 29, [114].TIME.MICROSECOND := 299842, [114].EVENT := '2016/06/29   09:53:29   FAULT : QOW1 : Charge Outside Window Detected', [115].TIME.YEAR := 2016, [115].TIME.MONTH := 6, [115].TIME.DAY := 29, [115].TIME.HOUR := 10, [115].TIME.MINUTE := 24, [115].TIME.SECOND := 10, [115].TIME.MICROSECOND := 199512, [115].EVENT := '2016/06/29   10:24:10   USER : PPS RESET FAULT BUTTON PRESSED', [116].TIME.YEAR := 2016, [116].TIME.MONTH := 6, [116].TIME.DAY := 29, [116].TIME.HOUR := 10, [116].TIME.MINUTE := 24, [116].TIME.SECOND := 14, [116].TIME.MICROSECOND := 600019, [116].EVENT := '2016/06/29   10:24:14   USER : PPS RESET FAULT BUTTON PRESSED', [117].TIME.YEAR := 2016, [117].TIME.MONTH := 6, [117].TIME.DAY := 29, [117].TIME.HOUR := 10, [117].TIME.MINUTE := 47, [117].TIME.SECOND := 33, [117].TIME.MICROSECOND := 199464, [117].EVENT := '2016/06/29   10:47:33   FAULT : QOW1 : Charge Outside Window Detected', [118].TIME.YEAR := 2016, [118].TIME.MONTH := 6, [118].TIME.DAY := 29, [118].TIME.HOUR := 11, [118].TIME.MINUTE := 41, [118].TIME.SECOND := 52, [118].TIME.MICROSECOND := 999507, [118].EVENT := '2016/06/29   11:41:52   USER : PPS RESET FAULT BUTTON PRESSED', [119].TIME.YEAR := 2016, [119].TIME.MONTH := 6, [119].TIME.DAY := 29, [119].TIME.HOUR := 14, [119].TIME.MINUTE := 41, [119].TIME.SECOND := 50, [119].TIME.MICROSECOND := 799510, [119].EVENT := '2016/06/29   14:41:50   USER : PPS RESET FAULT BUTTON PRESSED', [120].TIME.YEAR := 2016, [120].TIME.MONTH := 6, [120].TIME.DAY := 29, [120].TIME.HOUR := 15, [120].TIME.MINUTE := 26, [120].TIME.SECOND := 26, [120].TIME.MICROSECOND := 399719,
        [120].EVENT := '2016/06/29   15:26:26   USER : PPS RESET FAULT BUTTON PRESSED', [121].TIME.YEAR := 2016, [121].TIME.MONTH := 6, [121].TIME.DAY := 29, [121].TIME.HOUR := 16, [121].TIME.MINUTE := 17, [121].TIME.SECOND := 39, [121].TIME.MICROSECOND := 799507, [121].EVENT := '2016/06/29   16:17:39   USER : PPS RESET FAULT BUTTON PRESSED', [122].TIME.YEAR := 2016, [122].TIME.MONTH := 6, [122].TIME.DAY := 29, [122].TIME.HOUR := 16, [122].TIME.MINUTE := 17, [122].TIME.SECOND := 40, [122].TIME.MICROSECOND := 499513, [122].EVENT := '2016/06/29   16:17:40   USER : PPS RESET FAULT BUTTON PRESSED', [123].TIME.YEAR := 2016, [123].TIME.MONTH := 6, [123].TIME.DAY := 29, [123].TIME.HOUR := 17, [123].TIME.MINUTE := 21, [123].TIME.SECOND := 27, [123].TIME.MICROSECOND := 599509, [123].EVENT := '2016/06/29   17:21:27   FAULT : QOW1 : Charge Outside Window Detected', [124].TIME.YEAR := 2016, [124].TIME.MONTH := 6, [124].TIME.DAY := 29, [124].TIME.HOUR := 17, [124].TIME.MINUTE := 22, [124].TIME.SECOND := 46, [124].TIME.MICROSECOND := 599514, [124].EVENT := '2016/06/29   17:22:46   USER : PPS RESET FAULT BUTTON PRESSED', [125].TIME.YEAR := 2016, [125].TIME.MONTH := 6, [125].TIME.DAY := 30, [125].TIME.HOUR := 5, [125].TIME.MINUTE := 30, [125].TIME.SECOND := 17, [125].TIME.MICROSECOND := 299462, [125].EVENT := '2016/06/30   05:30:17   FAULT : QOW1 : Charge Outside Window Detected', [126].TIME.YEAR := 2016, [126].TIME.MONTH := 6, [126].TIME.DAY := 30, [126].TIME.HOUR := 5, [126].TIME.MINUTE := 31, [126].TIME.SECOND := 43, [126].TIME.MICROSECOND := 199511, [126].EVENT := '2016/06/30   05:31:43   USER : PPS RESET FAULT BUTTON PRESSED', [127].TIME.YEAR := 2016, [127].TIME.MONTH := 6, [127].TIME.DAY := 30, [127].TIME.HOUR := 5, [127].TIME.MINUTE := 31, [127].TIME.SECOND := 50, [127].TIME.MICROSECOND := 999516, [127].EVENT := '2016/06/30   05:31:50   USER : PPS RESET FAULT BUTTON PRESSED', [128].TIME.YEAR := 2016, [128].TIME.MONTH := 6, [128].TIME.DAY := 30,
        [128].TIME.HOUR := 5, [128].TIME.MINUTE := 47, [128].TIME.SECOND := 21, [128].TIME.MICROSECOND := 499940, [128].EVENT := '2016/06/30   05:47:21   USER : PPS RESET FAULT BUTTON PRESSED', [129].TIME.YEAR := 2016, [129].TIME.MONTH := 6, [129].TIME.DAY := 30, [129].TIME.HOUR := 5, [129].TIME.MINUTE := 48, [129].TIME.SECOND := 12, [129].TIME.MICROSECOND := 199513, [129].EVENT := '2016/06/30   05:48:12   USER : PPS RESET FAULT BUTTON PRESSED', [130].TIME.YEAR := 2016, [130].TIME.MONTH := 6, [130].TIME.DAY := 30, [130].TIME.HOUR := 5, [130].TIME.MINUTE := 48, [130].TIME.SECOND := 42, [130].TIME.MICROSECOND := 699503, [130].EVENT := '2016/06/30   05:48:42   USER : PPS RESET FAULT BUTTON PRESSED', [131].TIME.YEAR := 2016, [131].TIME.MONTH := 6, [131].TIME.DAY := 30, [131].TIME.HOUR := 6, [131].TIME.MINUTE := 58, [131].TIME.SECOND := 4, [131].TIME.MICROSECOND := 700021, [131].EVENT := '2016/06/30   06:58:04   USER : PPS RESET FAULT BUTTON PRESSED', [132].TIME.YEAR := 2016, [132].TIME.MONTH := 7, [132].TIME.DAY := 1, [132].TIME.HOUR := 19, [132].TIME.MINUTE := 23, [132].TIME.SECOND := 54, [132].TIME.MICROSECOND := 99506, [132].EVENT := '2016/07/01   19:23:54   USER : PPS RESET FAULT BUTTON PRESSED', [133].TIME.YEAR := 2016, [133].TIME.MONTH := 7, [133].TIME.DAY := 1, [133].TIME.HOUR := 19, [133].TIME.MINUTE := 23, [133].TIME.SECOND := 56, [133].TIME.MICROSECOND := 999506, [133].EVENT := '2016/07/01   19:23:56   USER : PPS RESET FAULT BUTTON PRESSED', [134].TIME.YEAR := 2016, [134].TIME.MONTH := 7, [134].TIME.DAY := 1, [134].TIME.HOUR := 19, [134].TIME.MINUTE := 24, [134].TIME.SECOND := 20, [134].TIME.MICROSECOND := 499522, [134].EVENT := '2016/07/01   19:24:20   USER : PPS RESET FAULT BUTTON PRESSED', [135].TIME.YEAR := 2016, [135].TIME.MONTH := 7, [135].TIME.DAY := 1, [135].TIME.HOUR := 19, [135].TIME.MINUTE := 24, [135].TIME.SECOND := 20, [135].TIME.MICROSECOND := 999468,
        [135].EVENT := '2016/07/01   19:24:20   FAULT : QOW1 : Charge Outside Window Detected', [136].TIME.YEAR := 2016, [136].TIME.MONTH := 7, [136].TIME.DAY := 1, [136].TIME.HOUR := 19, [136].TIME.MINUTE := 24, [136].TIME.SECOND := 21, [136].TIME.MICROSECOND := 99502, [136].EVENT := '2016/07/01   19:24:21   USER : PPS RESET FAULT BUTTON PRESSED', [137].TIME.YEAR := 2016, [137].TIME.MONTH := 7, [137].TIME.DAY := 1, [137].TIME.HOUR := 19, [137].TIME.MINUTE := 47, [137].TIME.SECOND := 12, [137].TIME.MICROSECOND := 800022, [137].EVENT := '2016/07/01   19:47:12   USER : PPS RESET FAULT BUTTON PRESSED', [138].TIME.YEAR := 2016, [138].TIME.MONTH := 7, [138].TIME.DAY := 1, [138].TIME.HOUR := 20, [138].TIME.MINUTE := 15, [138].TIME.SECOND := 15, [138].TIME.MICROSECOND := 99505, [138].EVENT := '2016/07/01   20:15:15   USER : PPS RESET FAULT BUTTON PRESSED', [139].TIME.YEAR := 2016, [139].TIME.MONTH := 7, [139].TIME.DAY := 1, [139].TIME.HOUR := 20, [139].TIME.MINUTE := 29, [139].TIME.SECOND := 50, [139].TIME.MICROSECOND := 200027, [139].EVENT := '2016/07/01   20:29:50   USER : PPS RESET FAULT BUTTON PRESSED', [140].TIME.YEAR := 2016, [140].TIME.MONTH := 7, [140].TIME.DAY := 1, [140].TIME.HOUR := 20, [140].TIME.MINUTE := 29, [140].TIME.SECOND := 51, [140].TIME.MICROSECOND := 999507, [140].EVENT := '2016/07/01   20:29:51   USER : PPS RESET FAULT BUTTON PRESSED', [141].TIME.YEAR := 2016, [141].TIME.MONTH := 7, [141].TIME.DAY := 1, [141].TIME.HOUR := 20, [141].TIME.MINUTE := 42, [141].TIME.SECOND := 22, [141].TIME.MICROSECOND := 999513, [141].EVENT := '2016/07/01   20:42:22   USER : PPS RESET FAULT BUTTON PRESSED', [142].TIME.YEAR := 2016, [142].TIME.MONTH := 7, [142].TIME.DAY := 3, [142].TIME.HOUR := 11, [142].TIME.MINUTE := 51, [142].TIME.SECOND := 18, [142].TIME.MICROSECOND := 599461, [142].EVENT := '2016/07/03   11:51:18   FAULT : Storage Ring Accumulation HIGH', [143].TIME.YEAR := 2016, [143].TIME.MONTH := 7, [143].TIME.DAY := 3,
        [143].TIME.HOUR := 11, [143].TIME.MINUTE := 51, [143].TIME.SECOND := 37, [143].TIME.MICROSECOND := 499453, [143].EVENT := '2016/07/03   11:51:37   FAULT : Storage Ring Accumulation HIGH', [144].TIME.YEAR := 2016, [144].TIME.MONTH := 7, [144].TIME.DAY := 3, [144].TIME.HOUR := 11, [144].TIME.MINUTE := 51, [144].TIME.SECOND := 38, [144].TIME.MICROSECOND := 99511, [144].EVENT := '2016/07/03   11:51:38   USER : PPS RESET FAULT BUTTON PRESSED', [145].TIME.YEAR := 2016, [145].TIME.MONTH := 7, [145].TIME.DAY := 3, [145].TIME.HOUR := 11, [145].TIME.MINUTE := 52, [145].TIME.SECOND := 3, [145].TIME.MICROSECOND := 899455, [145].EVENT := '2016/07/03   11:52:03   FAULT : Storage Ring Accumulation HIGH', [146].TIME.YEAR := 2016, [146].TIME.MONTH := 7, [146].TIME.DAY := 3, [146].TIME.HOUR := 11, [146].TIME.MINUTE := 52, [146].TIME.SECOND := 3, [146].TIME.MICROSECOND := 900059, [146].EVENT := '2016/07/03   11:52:03   USER : PPS RESET FAULT BUTTON PRESSED', [147].TIME.YEAR := 2016, [147].TIME.MONTH := 7, [147].TIME.DAY := 3, [147].TIME.HOUR := 11, [147].TIME.MINUTE := 52, [147].TIME.SECOND := 6, [147].TIME.MICROSECOND := 999453, [147].EVENT := '2016/07/03   11:52:06   FAULT : Storage Ring Accumulation HIGH', [148].TIME.YEAR := 2016, [148].TIME.MONTH := 7, [148].TIME.DAY := 3, [148].TIME.HOUR := 11, [148].TIME.MINUTE := 52, [148].TIME.SECOND := 8, [148].TIME.MICROSECOND := 99511, [148].EVENT := '2016/07/03   11:52:08   USER : PPS RESET FAULT BUTTON PRESSED', [149].TIME.YEAR := 2016, [149].TIME.MONTH := 7, [149].TIME.DAY := 3, [149].TIME.HOUR := 11, [149].TIME.MINUTE := 53, [149].TIME.SECOND := 31, [149].TIME.MICROSECOND := 499505, [149].EVENT := '2016/07/03   11:53:31   USER : PPS RESET FAULT BUTTON PRESSED', [150].TIME.YEAR := 2016, [150].TIME.MONTH := 7, [150].TIME.DAY := 3, [150].TIME.HOUR := 11, [150].TIME.MINUTE := 54, [150].TIME.SECOND := 55, [150].TIME.MICROSECOND := 599450,
        [150].EVENT := '2016/07/03   11:54:55   FAULT : Storage Ring Accumulation HIGH', [151].TIME.YEAR := 2016, [151].TIME.MONTH := 7, [151].TIME.DAY := 3, [151].TIME.HOUR := 11, [151].TIME.MINUTE := 55, [151].TIME.SECOND := 46, [151].TIME.MICROSECOND := 999502, [151].EVENT := '2016/07/03   11:55:46   USER : PPS RESET FAULT BUTTON PRESSED', [152].TIME.YEAR := 2016, [152].TIME.MONTH := 7, [152].TIME.DAY := 3, [152].TIME.HOUR := 11, [152].TIME.MINUTE := 57, [152].TIME.SECOND := 31, [152].TIME.MICROSECOND := 499454, [152].EVENT := '2016/07/03   11:57:31   FAULT : Storage Ring Accumulation HIGH', [153].TIME.YEAR := 2016, [153].TIME.MONTH := 7, [153].TIME.DAY := 3, [153].TIME.HOUR := 11, [153].TIME.MINUTE := 57, [153].TIME.SECOND := 31, [153].TIME.MICROSECOND := 699464, [153].EVENT := '2016/07/03   11:57:31   FAULT : QOW1 : Charge Outside Window Detected', [154].TIME.YEAR := 2016, [154].TIME.MONTH := 7, [154].TIME.DAY := 3, [154].TIME.HOUR := 11, [154].TIME.MINUTE := 58, [154].TIME.SECOND := 4, [154].TIME.MICROSECOND := 599507, [154].EVENT := '2016/07/03   11:58:04   USER : PPS RESET FAULT BUTTON PRESSED', [155].TIME.YEAR := 2016, [155].TIME.MONTH := 7, [155].TIME.DAY := 3, [155].TIME.HOUR := 12, [155].TIME.SECOND := 13, [155].TIME.MICROSECOND := 499449, [155].EVENT := '2016/07/03   12:00:13   FAULT : Storage Ring Accumulation HIGH', [156].TIME.YEAR := 2016, [156].TIME.MONTH := 7, [156].TIME.DAY := 3, [156].TIME.HOUR := 12, [156].TIME.SECOND := 46, [156].TIME.MICROSECOND := 699509, [156].EVENT := '2016/07/03   12:00:46   USER : PPS RESET FAULT BUTTON PRESSED', [157].TIME.YEAR := 2016, [157].TIME.MONTH := 7, [157].TIME.DAY := 5, [157].TIME.HOUR := 10, [157].TIME.MINUTE := 55, [157].TIME.SECOND := 24, [157].TIME.MICROSECOND := 399722, [157].EVENT := '2016/07/05   10:55:24   USER : PPS RESET FAULT BUTTON PRESSED', [158].TIME.YEAR := 2016, [158].TIME.MONTH := 7, [158].TIME.DAY := 6, [158].TIME.HOUR := 14, [158].TIME.MINUTE := 34,
        [158].TIME.SECOND := 52, [158].TIME.MICROSECOND := 299939, [158].EVENT := '2016/07/06   14:34:52   USER : PPS RESET FAULT BUTTON PRESSED', [159].TIME.YEAR := 2016, [159].TIME.MONTH := 7, [159].TIME.DAY := 6, [159].TIME.HOUR := 18, [159].TIME.MINUTE := 37, [159].TIME.SECOND := 59, [159].TIME.MICROSECOND := 200096, [159].EVENT := '2016/07/06   18:37:59   USER : PPS RESET FAULT BUTTON PRESSED', [160].TIME.YEAR := 2016, [160].TIME.MONTH := 7, [160].TIME.DAY := 6, [160].TIME.HOUR := 18, [160].TIME.MINUTE := 38, [160].TIME.SECOND := 2, [160].TIME.MICROSECOND := 499508, [160].EVENT := '2016/07/06   18:38:02   USER : PPS RESET FAULT BUTTON PRESSED', [161].TIME.YEAR := 2016, [161].TIME.MONTH := 7, [161].TIME.DAY := 7, [161].TIME.MINUTE := 27, [161].TIME.SECOND := 18, [161].TIME.MICROSECOND := 699513, [161].EVENT := '2016/07/07   00:27:18   USER : PPS RESET FAULT BUTTON PRESSED', [162].TIME.YEAR := 2016, [162].TIME.MONTH := 7, [162].TIME.DAY := 7, [162].TIME.MINUTE := 27, [162].TIME.SECOND := 21, [162].TIME.MICROSECOND := 699512, [162].EVENT := '2016/07/07   00:27:21   USER : PPS RESET FAULT BUTTON PRESSED', [163].TIME.YEAR := 2016, [163].TIME.MONTH := 7, [163].TIME.DAY := 7, [163].TIME.MINUTE := 38, [163].TIME.SECOND := 50, [163].TIME.MICROSECOND := 399510, [163].EVENT := '2016/07/07   00:38:50   USER : PPS RESET FAULT BUTTON PRESSED', [164].TIME.YEAR := 2016, [164].TIME.MONTH := 7, [164].TIME.DAY := 7, [164].TIME.HOUR := 8, [164].TIME.MINUTE := 1, [164].TIME.SECOND := 39, [164].TIME.MICROSECOND := 599463, [164].EVENT := '2016/07/07   08:01:39   FAULT : QOW1 : Charge Outside Window Detected', [165].TIME.YEAR := 2016, [165].TIME.MONTH := 7, [165].TIME.DAY := 7, [165].TIME.HOUR := 8, [165].TIME.MINUTE := 4, [165].TIME.SECOND := 34, [165].TIME.MICROSECOND := 199509, [165].EVENT := '2016/07/07   08:04:34   USER : PPS RESET FAULT BUTTON PRESSED', [166].TIME.YEAR := 2016, [166].TIME.MONTH := 7, [166].TIME.DAY := 7, [166].TIME.HOUR := 8,
        [166].TIME.MINUTE := 20, [166].TIME.SECOND := 42, [166].TIME.MICROSECOND := 799509, [166].EVENT := '2016/07/07   08:20:42   USER : PPS RESET FAULT BUTTON PRESSED', [167].TIME.YEAR := 2016, [167].TIME.MONTH := 7, [167].TIME.DAY := 7, [167].TIME.HOUR := 14, [167].TIME.MINUTE := 52, [167].TIME.SECOND := 49, [167].TIME.MICROSECOND := 599517, [167].EVENT := '2016/07/07   14:52:49   USER : PPS RESET FAULT BUTTON PRESSED', [168].TIME.YEAR := 2016, [168].TIME.MONTH := 7, [168].TIME.DAY := 8, [168].TIME.HOUR := 7, [168].TIME.MINUTE := 10, [168].TIME.SECOND := 26, [168].TIME.MICROSECOND := 699554, [168].EVENT := '2016/07/08   07:10:26   USER : PPS RESET FAULT BUTTON PRESSED', [169].TIME.YEAR := 2016, [169].TIME.MONTH := 7, [169].TIME.DAY := 9, [169].TIME.HOUR := 12, [169].TIME.MINUTE := 14, [169].TIME.SECOND := 28, [169].TIME.MICROSECOND := 99584, [169].EVENT := '2016/07/09   12:14:28   FAULT : QOW1 : Charge Outside Window Detected', [170].TIME.YEAR := 2016, [170].TIME.MONTH := 7, [170].TIME.DAY := 9, [170].TIME.HOUR := 12, [170].TIME.MINUTE := 14, [170].TIME.SECOND := 28, [170].TIME.MICROSECOND := 399524, [170].EVENT := '2016/07/09   12:14:28   USER : PPS RESET FAULT BUTTON PRESSED', [171].TIME.YEAR := 2016, [171].TIME.MONTH := 7, [171].TIME.DAY := 9, [171].TIME.HOUR := 12, [171].TIME.MINUTE := 15, [171].TIME.SECOND := 1, [171].TIME.MICROSECOND := 199506, [171].EVENT := '2016/07/09   12:15:01   USER : PPS RESET FAULT BUTTON PRESSED', [172].TIME.YEAR := 2016, [172].TIME.MONTH := 7, [172].TIME.DAY := 9, [172].TIME.HOUR := 14, [172].TIME.MINUTE := 35, [172].TIME.SECOND := 17, [172].TIME.MICROSECOND := 299510, [172].EVENT := '2016/07/09   14:35:17   USER : PPS RESET FAULT BUTTON PRESSED', [173].TIME.YEAR := 2016, [173].TIME.MONTH := 7, [173].TIME.DAY := 9, [173].TIME.HOUR := 14, [173].TIME.MINUTE := 35, [173].TIME.SECOND := 52, [173].TIME.MICROSECOND := 499458, [173].EVENT := '2016/07/09   14:35:52   FAULT : QOW1 : Charge Outside Window Detected',
        [174].TIME.YEAR := 2016, [174].TIME.MONTH := 7, [174].TIME.DAY := 9, [174].TIME.HOUR := 14, [174].TIME.MINUTE := 36, [174].TIME.SECOND := 10, [174].TIME.MICROSECOND := 799512, [174].EVENT := '2016/07/09   14:36:10   USER : PPS RESET FAULT BUTTON PRESSED', [175].TIME.YEAR := 2016, [175].TIME.MONTH := 7, [175].TIME.DAY := 9, [175].TIME.HOUR := 14, [175].TIME.MINUTE := 50, [175].TIME.SECOND := 4, [175].TIME.MICROSECOND := 100155, [175].EVENT := '2016/07/09   14:50:04   USER : PPS RESET FAULT BUTTON PRESSED', [176].TIME.YEAR := 2016, [176].TIME.MONTH := 7, [176].TIME.DAY := 10, [176].TIME.HOUR := 14, [176].TIME.MINUTE := 2, [176].TIME.SECOND := 1, [176].TIME.MICROSECOND := 299504, [176].EVENT := '2016/07/10   14:02:01   USER : PPS RESET FAULT BUTTON PRESSED', [177].TIME.YEAR := 2016, [177].TIME.MONTH := 7, [177].TIME.DAY := 10, [177].TIME.HOUR := 14, [177].TIME.MINUTE := 2, [177].TIME.SECOND := 6, [177].TIME.MICROSECOND := 399509, [177].EVENT := '2016/07/10   14:02:06   USER : PPS RESET FAULT BUTTON PRESSED', [178].TIME.YEAR := 2016, [178].TIME.MONTH := 7, [178].TIME.DAY := 10, [178].TIME.HOUR := 15, [178].TIME.MINUTE := 17, [178].TIME.SECOND := 47, [178].TIME.MICROSECOND := 799549, [178].EVENT := '2016/07/10   15:17:47   USER : PPS RESET FAULT BUTTON PRESSED', [179].TIME.YEAR := 2016, [179].TIME.MONTH := 7, [179].TIME.DAY := 10, [179].TIME.HOUR := 15, [179].TIME.MINUTE := 24, [179].TIME.SECOND := 7, [179].TIME.MICROSECOND := 199510, [179].EVENT := '2016/07/10   15:24:07   USER : PPS RESET FAULT BUTTON PRESSED', [180].TIME.YEAR := 2016, [180].TIME.MONTH := 7, [180].TIME.DAY := 10, [180].TIME.HOUR := 15, [180].TIME.MINUTE := 49, [180].TIME.SECOND := 42, [180].TIME.MICROSECOND := 499515, [180].EVENT := '2016/07/10   15:49:42   USER : PPS RESET FAULT BUTTON PRESSED', [181].TIME.YEAR := 2016, [181].TIME.MONTH := 7, [181].TIME.DAY := 10, [181].TIME.HOUR := 15,
        [181].TIME.MINUTE := 49, [181].TIME.SECOND := 53, [181].TIME.MICROSECOND := 99938, [181].EVENT := '2016/07/10   15:49:53   USER : PPS RESET FAULT BUTTON PRESSED', [182].TIME.YEAR := 2016, [182].TIME.MONTH := 7, [182].TIME.DAY := 10, [182].TIME.HOUR := 16, [182].TIME.MINUTE := 45, [182].TIME.SECOND := 14, [182].TIME.MICROSECOND := 299509, [182].EVENT := '2016/07/10   16:45:14   USER : PPS RESET FAULT BUTTON PRESSED', [183].TIME.YEAR := 2016, [183].TIME.MONTH := 7, [183].TIME.DAY := 10, [183].TIME.HOUR := 16, [183].TIME.MINUTE := 49, [183].TIME.SECOND := 52, [183].TIME.MICROSECOND := 99691, [183].EVENT := '2016/07/10   16:49:52   FAULT : QOW1 : Charge Outside Window Detected', [184].TIME.YEAR := 2016, [184].TIME.MONTH := 7, [184].TIME.DAY := 10, [184].TIME.HOUR := 16, [184].TIME.MINUTE := 50, [184].TIME.MICROSECOND := 199508, [184].EVENT := '2016/07/10   16:50:00   USER : PPS RESET FAULT BUTTON PRESSED', [185].TIME.YEAR := 2016, [185].TIME.MONTH := 7, [185].TIME.DAY := 11, [185].TIME.HOUR := 8, [185].TIME.MINUTE := 12, [185].TIME.SECOND := 26, [185].TIME.MICROSECOND := 499677, [185].EVENT := '2016/07/11   08:12:26   FAULT : QOW1 : Charge Outside Window Detected', [186].TIME.YEAR := 2016, [186].TIME.MONTH := 7, [186].TIME.DAY := 11, [186].TIME.HOUR := 8, [186].TIME.MINUTE := 34, [186].TIME.SECOND := 54, [186].TIME.MICROSECOND := 999509, [186].EVENT := '2016/07/11   08:34:54   USER : PPS RESET FAULT BUTTON PRESSED', [187].TIME.YEAR := 2016, [187].TIME.MONTH := 7, [187].TIME.DAY := 11, [187].TIME.HOUR := 10, [187].TIME.MINUTE := 28, [187].TIME.SECOND := 12, [187].TIME.MICROSECOND := 799463, [187].EVENT := '2016/07/11   10:28:12   FAULT : QOW1 : Charge Outside Window Detected', [188].TIME.YEAR := 2016, [188].TIME.MONTH := 7, [188].TIME.DAY := 11, [188].TIME.HOUR := 10, [188].TIME.MINUTE := 29, [188].TIME.SECOND := 17, [188].TIME.MICROSECOND := 599504, [188].EVENT := '2016/07/11   10:29:17   USER : PPS RESET FAULT BUTTON PRESSED', [189].TIME.YEAR := 2016,
        [189].TIME.MONTH := 7, [189].TIME.DAY := 11, [189].TIME.HOUR := 10, [189].TIME.MINUTE := 32, [189].TIME.SECOND := 35, [189].TIME.MICROSECOND := 299468, [189].EVENT := '2016/07/11   10:32:35   FAULT : QOW1 : Charge Outside Window Detected', [190].TIME.YEAR := 2016, [190].TIME.MONTH := 7, [190].TIME.DAY := 11, [190].TIME.HOUR := 10, [190].TIME.MINUTE := 32, [190].TIME.SECOND := 49, [190].TIME.MICROSECOND := 699512, [190].EVENT := '2016/07/11   10:32:49   USER : PPS RESET FAULT BUTTON PRESSED', [191].TIME.YEAR := 2016, [191].TIME.MONTH := 7, [191].TIME.DAY := 11, [191].TIME.HOUR := 10, [191].TIME.MINUTE := 32, [191].TIME.SECOND := 50, [191].TIME.MICROSECOND := 599509, [191].EVENT := '2016/07/11   10:32:50   USER : PPS RESET FAULT BUTTON PRESSED', [192].TIME.YEAR := 2016, [192].TIME.MONTH := 7, [192].TIME.DAY := 11, [192].TIME.HOUR := 10, [192].TIME.MINUTE := 36, [192].TIME.SECOND := 25, [192].TIME.MICROSECOND := 699584, [192].EVENT := '2016/07/11   10:36:25   USER : PPS RESET FAULT BUTTON PRESSED', [193].TIME.YEAR := 2016, [193].TIME.MONTH := 7, [193].TIME.DAY := 11, [193].TIME.HOUR := 10, [193].TIME.MINUTE := 36, [193].TIME.SECOND := 53, [193].TIME.MICROSECOND := 99507, [193].EVENT := '2016/07/11   10:36:53   USER : PPS RESET FAULT BUTTON PRESSED', [194].TIME.YEAR := 2016, [194].TIME.MONTH := 7, [194].TIME.DAY := 11, [194].TIME.HOUR := 10, [194].TIME.MINUTE := 36, [194].TIME.SECOND := 53, [194].TIME.MICROSECOND := 399942, [194].EVENT := '2016/07/11   10:36:53   USER : PPS RESET FAULT BUTTON PRESSED', [195].TIME.YEAR := 2016, [195].TIME.MONTH := 7, [195].TIME.DAY := 11, [195].TIME.HOUR := 10, [195].TIME.MINUTE := 51, [195].TIME.SECOND := 34, [195].TIME.MICROSECOND := 399506, [195].EVENT := '2016/07/11   10:51:34   USER : PPS RESET FAULT BUTTON PRESSED', [196].TIME.YEAR := 2016, [196].TIME.MONTH := 7, [196].TIME.DAY := 11, [196].TIME.HOUR := 11, [196].TIME.MINUTE := 17,
        [196].TIME.SECOND := 55, [196].TIME.MICROSECOND := 899510, [196].EVENT := '2016/07/11   11:17:55   USER : PPS RESET FAULT BUTTON PRESSED', [197].TIME.YEAR := 2016, [197].TIME.MONTH := 7, [197].TIME.DAY := 11, [197].TIME.HOUR := 11, [197].TIME.MINUTE := 30, [197].TIME.SECOND := 16, [197].TIME.MICROSECOND := 799941, [197].EVENT := '2016/07/11   11:30:16   USER : PPS RESET FAULT BUTTON PRESSED', [198].TIME.YEAR := 2016, [198].TIME.MONTH := 7, [198].TIME.DAY := 11, [198].TIME.HOUR := 11, [198].TIME.MINUTE := 30, [198].TIME.SECOND := 17, [198].TIME.MICROSECOND := 300040, [198].EVENT := '2016/07/11   11:30:17   USER : PPS RESET FAULT BUTTON PRESSED', [199].TIME.YEAR := 2016, [199].TIME.MONTH := 7, [199].TIME.DAY := 11, [199].TIME.HOUR := 11, [199].TIME.MINUTE := 37, [199].TIME.SECOND := 9, [199].TIME.MICROSECOND := 499464, [199].EVENT := '2016/07/11   11:37:09   FAULT : QOW1 : Charge Outside Window Detected', [200].TIME.YEAR := 2016, [200].TIME.MONTH := 7, [200].TIME.DAY := 11, [200].TIME.HOUR := 11, [200].TIME.MINUTE := 40, [200].TIME.SECOND := 10, [200].TIME.MICROSECOND := 300022, [200].EVENT := '2016/07/11   11:40:10   USER : PPS RESET FAULT BUTTON PRESSED', [201].TIME.YEAR := 2016, [201].TIME.MONTH := 7, [201].TIME.DAY := 11, [201].TIME.HOUR := 11, [201].TIME.MINUTE := 40, [201].TIME.SECOND := 10, [201].TIME.MICROSECOND := 899540, [201].EVENT := '2016/07/11   11:40:10   USER : PPS RESET FAULT BUTTON PRESSED', [202].TIME.YEAR := 2016, [202].TIME.MONTH := 7, [202].TIME.DAY := 11, [202].TIME.HOUR := 11, [202].TIME.MINUTE := 40, [202].TIME.SECOND := 11, [202].TIME.MICROSECOND := 99654, [202].EVENT := '2016/07/11   11:40:11   USER : PPS RESET FAULT BUTTON PRESSED', [203].TIME.YEAR := 2016, [203].TIME.MONTH := 7, [203].TIME.DAY := 11, [203].TIME.HOUR := 11, [203].TIME.MINUTE := 40, [203].TIME.SECOND := 11, [203].TIME.MICROSECOND := 399565, [203].EVENT := '2016/07/11   11:40:11   USER : PPS RESET FAULT BUTTON PRESSED', [204].TIME.YEAR := 2016,
        [204].TIME.MONTH := 7, [204].TIME.DAY := 11, [204].TIME.HOUR := 13, [204].TIME.MINUTE := 28, [204].TIME.SECOND := 32, [204].TIME.MICROSECOND := 99508, [204].EVENT := '2016/07/11   13:28:32   USER : PPS RESET FAULT BUTTON PRESSED', [205].TIME.YEAR := 2016, [205].TIME.MONTH := 7, [205].TIME.DAY := 11, [205].TIME.HOUR := 17, [205].TIME.MINUTE := 29, [205].TIME.SECOND := 6, [205].TIME.MICROSECOND := 799462, [205].EVENT := '2016/07/11   17:29:06   FAULT : QOW1 : Charge Outside Window Detected', [206].TIME.YEAR := 2016, [206].TIME.MONTH := 7, [206].TIME.DAY := 11, [206].TIME.HOUR := 17, [206].TIME.MINUTE := 29, [206].TIME.SECOND := 35, [206].TIME.MICROSECOND := 299509, [206].EVENT := '2016/07/11   17:29:35   USER : PPS RESET FAULT BUTTON PRESSED', [207].TIME.YEAR := 2016, [207].TIME.MONTH := 7, [207].TIME.DAY := 11, [207].TIME.HOUR := 17, [207].TIME.MINUTE := 30, [207].TIME.SECOND := 40, [207].TIME.MICROSECOND := 499513, [207].EVENT := '2016/07/11   17:30:40   USER : PPS RESET FAULT BUTTON PRESSED', [208].TIME.YEAR := 2016, [208].TIME.MONTH := 7, [208].TIME.DAY := 11, [208].TIME.HOUR := 17, [208].TIME.MINUTE := 37, [208].TIME.SECOND := 38, [208].TIME.MICROSECOND := 999507, [208].EVENT := '2016/07/11   17:37:38   USER : PPS RESET FAULT BUTTON PRESSED', [209].TIME.YEAR := 2016, [209].TIME.MONTH := 7, [209].TIME.DAY := 11, [209].TIME.HOUR := 17, [209].TIME.MINUTE := 37, [209].TIME.SECOND := 39, [209].TIME.MICROSECOND := 899508, [209].EVENT := '2016/07/11   17:37:39   USER : PPS RESET FAULT BUTTON PRESSED', [210].TIME.YEAR := 2016, [210].TIME.MONTH := 7, [210].TIME.DAY := 11, [210].TIME.HOUR := 17, [210].TIME.MINUTE := 37, [210].TIME.SECOND := 40, [210].TIME.MICROSECOND := 299508, [210].EVENT := '2016/07/11   17:37:40   USER : PPS RESET FAULT BUTTON PRESSED', [211].TIME.YEAR := 2016, [211].TIME.MONTH := 7, [211].TIME.DAY := 11, [211].TIME.HOUR := 18, [211].TIME.MINUTE := 5,
        [211].TIME.SECOND := 44, [211].TIME.MICROSECOND := 399506, [211].EVENT := '2016/07/11   18:05:44   USER : PPS RESET FAULT BUTTON PRESSED', [212].TIME.YEAR := 2016, [212].TIME.MONTH := 7, [212].TIME.DAY := 11, [212].TIME.HOUR := 18, [212].TIME.MINUTE := 43, [212].TIME.SECOND := 3, [212].TIME.MICROSECOND := 899505, [212].EVENT := '2016/07/11   18:43:03   USER : PPS RESET FAULT BUTTON PRESSED', [213].TIME.YEAR := 2016, [213].TIME.MONTH := 7, [213].TIME.DAY := 11, [213].TIME.HOUR := 19, [213].TIME.MINUTE := 12, [213].TIME.SECOND := 9, [213].TIME.MICROSECOND := 999505, [213].EVENT := '2016/07/11   19:12:09   USER : PPS RESET FAULT BUTTON PRESSED', [214].TIME.YEAR := 2016, [214].TIME.MONTH := 7, [214].TIME.DAY := 11, [214].TIME.HOUR := 19, [214].TIME.MINUTE := 15, [214].TIME.SECOND := 15, [214].TIME.MICROSECOND := 299536, [214].EVENT := '2016/07/11   19:15:15   FAULT : QOW1 : Charge Outside Window Detected', [215].TIME.YEAR := 2016, [215].TIME.MONTH := 7, [215].TIME.DAY := 11, [215].TIME.HOUR := 19, [215].TIME.MINUTE := 35, [215].TIME.SECOND := 25, [215].TIME.MICROSECOND := 999939, [215].EVENT := '2016/07/11   19:35:25   USER : PPS RESET FAULT BUTTON PRESSED', [216].TIME.YEAR := 2016, [216].TIME.MONTH := 7, [216].TIME.DAY := 12, [216].TIME.HOUR := 13, [216].TIME.MINUTE := 49, [216].TIME.SECOND := 13, [216].TIME.MICROSECOND := 999507, [216].EVENT := '2016/07/12   13:49:13   USER : PPS RESET FAULT BUTTON PRESSED', [217].TIME.YEAR := 2016, [217].TIME.MONTH := 7, [217].TIME.DAY := 12, [217].TIME.HOUR := 13, [217].TIME.MINUTE := 49, [217].TIME.SECOND := 18, [217].TIME.MICROSECOND := 899935, [217].EVENT := '2016/07/12   13:49:18   USER : PPS RESET FAULT BUTTON PRESSED', [218].TIME.YEAR := 2016, [218].TIME.MONTH := 7, [218].TIME.DAY := 12, [218].TIME.HOUR := 13, [218].TIME.MINUTE := 49, [218].TIME.SECOND := 25, [218].TIME.MICROSECOND := 99600, [218].EVENT := '2016/07/12   13:49:25   USER : PPS RESET FAULT BUTTON PRESSED', [219].TIME.YEAR := 2016,
        [219].TIME.MONTH := 7, [219].TIME.DAY := 12, [219].TIME.HOUR := 13, [219].TIME.MINUTE := 49, [219].TIME.SECOND := 32, [219].TIME.MICROSECOND := 399504, [219].EVENT := '2016/07/12   13:49:32   USER : PPS RESET FAULT BUTTON PRESSED', [220].TIME.YEAR := 2016, [220].TIME.MONTH := 7, [220].TIME.DAY := 12, [220].TIME.HOUR := 13, [220].TIME.MINUTE := 49, [220].TIME.SECOND := 53, [220].TIME.MICROSECOND := 199506, [220].EVENT := '2016/07/12   13:49:53   USER : PPS RESET FAULT BUTTON PRESSED', [221].TIME.YEAR := 2016, [221].TIME.MONTH := 7, [221].TIME.DAY := 12, [221].TIME.HOUR := 13, [221].TIME.MINUTE := 50, [221].TIME.SECOND := 2, [221].TIME.MICROSECOND := 599505, [221].EVENT := '2016/07/12   13:50:02   USER : PPS RESET FAULT BUTTON PRESSED', [222].TIME.YEAR := 2016, [222].TIME.MONTH := 7, [222].TIME.DAY := 12, [222].TIME.HOUR := 13, [222].TIME.MINUTE := 50, [222].TIME.SECOND := 53, [222].TIME.MICROSECOND := 999508, [222].EVENT := '2016/07/12   13:50:53   USER : PPS RESET FAULT BUTTON PRESSED', [223].TIME.YEAR := 2016, [223].TIME.MONTH := 7, [223].TIME.DAY := 12, [223].TIME.HOUR := 13, [223].TIME.MINUTE := 51, [223].TIME.SECOND := 14, [223].TIME.MICROSECOND := 899506, [223].EVENT := '2016/07/12   13:51:14   USER : PPS RESET FAULT BUTTON PRESSED', [224].TIME.YEAR := 2016, [224].TIME.MONTH := 7, [224].TIME.DAY := 12, [224].TIME.HOUR := 13, [224].TIME.MINUTE := 51, [224].TIME.SECOND := 47, [224].TIME.MICROSECOND := 599944, [224].EVENT := '2016/07/12   13:51:47   USER : PPS RESET FAULT BUTTON PRESSED', [225].TIME.YEAR := 2016, [225].TIME.MONTH := 7, [225].TIME.DAY := 12, [225].TIME.HOUR := 13, [225].TIME.MINUTE := 52, [225].TIME.MICROSECOND := 199508, [225].EVENT := '2016/07/12   13:52:00   USER : PPS RESET FAULT BUTTON PRESSED', [226].TIME.YEAR := 2016, [226].TIME.MONTH := 7, [226].TIME.DAY := 12, [226].TIME.HOUR := 13, [226].TIME.MINUTE := 52, [226].TIME.SECOND := 4,
        [226].TIME.MICROSECOND := 599558, [226].EVENT := '2016/07/12   13:52:04   USER : PPS RESET FAULT BUTTON PRESSED', [227].TIME.YEAR := 2016, [227].TIME.MONTH := 7, [227].TIME.DAY := 12, [227].TIME.HOUR := 13, [227].TIME.MINUTE := 52, [227].TIME.SECOND := 16, [227].TIME.MICROSECOND := 199578, [227].EVENT := '2016/07/12   13:52:16   USER : PPS RESET FAULT BUTTON PRESSED', [228].TIME.YEAR := 2016, [228].TIME.MONTH := 7, [228].TIME.DAY := 12, [228].TIME.HOUR := 13, [228].TIME.MINUTE := 52, [228].TIME.SECOND := 19, [228].TIME.MICROSECOND := 299504, [228].EVENT := '2016/07/12   13:52:19   USER : PPS RESET FAULT BUTTON PRESSED', [229].TIME.YEAR := 2016, [229].TIME.MONTH := 7, [229].TIME.DAY := 12, [229].TIME.HOUR := 13, [229].TIME.MINUTE := 52, [229].TIME.SECOND := 21, [229].TIME.MICROSECOND := 200027, [229].EVENT := '2016/07/12   13:52:21   USER : PPS RESET FAULT BUTTON PRESSED', [230].TIME.YEAR := 2016, [230].TIME.MONTH := 7, [230].TIME.DAY := 12, [230].TIME.HOUR := 13, [230].TIME.MINUTE := 53, [230].TIME.SECOND := 9, [230].TIME.MICROSECOND := 799505, [230].EVENT := '2016/07/12   13:53:09   USER : PPS RESET FAULT BUTTON PRESSED', [231].TIME.YEAR := 2016, [231].TIME.MONTH := 7, [231].TIME.DAY := 12, [231].TIME.HOUR := 13, [231].TIME.MINUTE := 53, [231].TIME.SECOND := 40, [231].TIME.MICROSECOND := 799506, [231].EVENT := '2016/07/12   13:53:40   USER : PPS RESET FAULT BUTTON PRESSED', [232].TIME.YEAR := 2016, [232].TIME.MONTH := 7, [232].TIME.DAY := 12, [232].TIME.HOUR := 15, [232].TIME.MINUTE := 59, [232].TIME.SECOND := 48, [232].TIME.MICROSECOND := 199466, [232].EVENT := '2016/07/12   15:59:48   FAULT : QOW1 : Charge Outside Window Detected', [233].TIME.YEAR := 2016, [233].TIME.MONTH := 7, [233].TIME.DAY := 12, [233].TIME.HOUR := 18, [233].TIME.MINUTE := 2, [233].TIME.SECOND := 55, [233].TIME.MICROSECOND := 499936, [233].EVENT := '2016/07/12   18:02:55   USER : PPS RESET FAULT BUTTON PRESSED', [234].TIME.YEAR := 2016, [234].TIME.MONTH := 7,
        [234].TIME.DAY := 12, [234].TIME.HOUR := 20, [234].TIME.MINUTE := 9, [234].TIME.SECOND := 37, [234].TIME.MICROSECOND := 599509, [234].EVENT := '2016/07/12   20:09:37   USER : PPS RESET FAULT BUTTON PRESSED', [235].TIME.YEAR := 2016, [235].TIME.MONTH := 7, [235].TIME.DAY := 13, [235].TIME.HOUR := 11, [235].TIME.MINUTE := 45, [235].TIME.SECOND := 36, [235].TIME.MICROSECOND := 99652, [235].EVENT := '2016/07/13   11:45:36   USER : PPS RESET FAULT BUTTON PRESSED', [236].TIME.YEAR := 2016, [236].TIME.MONTH := 7, [236].TIME.DAY := 13, [236].TIME.HOUR := 11, [236].TIME.MINUTE := 59, [236].TIME.SECOND := 18, [236].TIME.MICROSECOND := 499466, [236].EVENT := '2016/07/13   11:59:18   FAULT : QOW1 : Charge Outside Window Detected', [237].TIME.YEAR := 2016, [237].TIME.MONTH := 7, [237].TIME.DAY := 13, [237].TIME.HOUR := 12, [237].TIME.MINUTE := 50, [237].TIME.SECOND := 31, [237].TIME.MICROSECOND := 799506, [237].EVENT := '2016/07/13   12:50:31   USER : PPS RESET FAULT BUTTON PRESSED', [238].TIME.YEAR := 2016, [238].TIME.MONTH := 7, [238].TIME.DAY := 13, [238].TIME.HOUR := 16, [238].TIME.MINUTE := 58, [238].TIME.SECOND := 29, [238].TIME.MICROSECOND := 199939, [238].EVENT := '2016/07/13   16:58:29   USER : PPS RESET FAULT BUTTON PRESSED', [239].TIME.YEAR := 2016, [239].TIME.MONTH := 7, [239].TIME.DAY := 13, [239].TIME.HOUR := 17, [239].TIME.MINUTE := 8, [239].TIME.SECOND := 56, [239].TIME.MICROSECOND := 299508, [239].EVENT := '2016/07/13   17:08:56   USER : PPS RESET FAULT BUTTON PRESSED', [240].TIME.YEAR := 2016, [240].TIME.MONTH := 7, [240].TIME.DAY := 13, [240].TIME.HOUR := 17, [240].TIME.MINUTE := 31, [240].TIME.SECOND := 47, [240].TIME.MICROSECOND := 199557, [240].EVENT := '2016/07/13   17:31:47   USER : PPS RESET FAULT BUTTON PRESSED', [241].TIME.YEAR := 2016, [241].TIME.MONTH := 7, [241].TIME.DAY := 13, [241].TIME.HOUR := 18, [241].TIME.MINUTE := 4, [241].TIME.SECOND := 28,
        [241].TIME.MICROSECOND := 999508, [241].EVENT := '2016/07/13   18:04:28   USER : PPS RESET FAULT BUTTON PRESSED', [242].TIME.YEAR := 2016, [242].TIME.MONTH := 7, [242].TIME.DAY := 13, [242].TIME.HOUR := 18, [242].TIME.MINUTE := 21, [242].TIME.SECOND := 13, [242].TIME.MICROSECOND := 999503, [242].EVENT := '2016/07/13   18:21:13   USER : PPS RESET FAULT BUTTON PRESSED', [243].TIME.YEAR := 2016, [243].TIME.MONTH := 7, [243].TIME.DAY := 13, [243].TIME.HOUR := 18, [243].TIME.MINUTE := 33, [243].TIME.SECOND := 34, [243].TIME.MICROSECOND := 799513, [243].EVENT := '2016/07/13   18:33:34   USER : PPS RESET FAULT BUTTON PRESSED', [244].TIME.YEAR := 2016, [244].TIME.MONTH := 7, [244].TIME.DAY := 13, [244].TIME.HOUR := 18, [244].TIME.MINUTE := 37, [244].TIME.SECOND := 2, [244].TIME.MICROSECOND := 799556, [244].EVENT := '2016/07/13   18:37:02   USER : PPS RESET FAULT BUTTON PRESSED', [245].TIME.YEAR := 2016, [245].TIME.MONTH := 7, [245].TIME.DAY := 14, [245].TIME.HOUR := 3, [245].TIME.MINUTE := 15, [245].TIME.SECOND := 27, [245].TIME.MICROSECOND := 999531, [245].EVENT := '2016/07/14   03:15:27   USER : PPS RESET FAULT BUTTON PRESSED', [246].TIME.YEAR := 2016, [246].TIME.MONTH := 7, [246].TIME.DAY := 14, [246].TIME.HOUR := 6, [246].TIME.MINUTE := 51, [246].TIME.SECOND := 54, [246].TIME.MICROSECOND := 99507, [246].EVENT := '2016/07/14   06:51:54   USER : PPS RESET FAULT BUTTON PRESSED', [247].TIME.YEAR := 2016, [247].TIME.MONTH := 7, [247].TIME.DAY := 15, [247].TIME.HOUR := 6, [247].TIME.MINUTE := 39, [247].TIME.SECOND := 41, [247].TIME.MICROSECOND := 999465, [247].EVENT := '2016/07/15   06:39:41   FAULT : QOW1 : Charge Outside Window Detected', [248].TIME.YEAR := 2016, [248].TIME.MONTH := 7, [248].TIME.DAY := 15, [248].TIME.HOUR := 6, [248].TIME.MINUTE := 53, [248].TIME.SECOND := 26, [248].TIME.MICROSECOND := 299508, [248].EVENT := '2016/07/15   06:53:26   USER : PPS RESET FAULT BUTTON PRESSED', [249].TIME.YEAR := 2016, [249].TIME.MONTH := 7,
        [249].TIME.DAY := 16, [249].TIME.HOUR := 9, [249].TIME.MINUTE := 29, [249].TIME.SECOND := 54, [249].TIME.MICROSECOND := 999509, [249].EVENT := '2016/07/16   09:29:54   USER : PPS RESET FAULT BUTTON PRESSED', [250].TIME.YEAR := 2016, [250].TIME.MONTH := 7, [250].TIME.DAY := 16, [250].TIME.HOUR := 9, [250].TIME.MINUTE := 47, [250].TIME.SECOND := 17, [250].TIME.MICROSECOND := 299468, [250].EVENT := '2016/07/16   09:47:17   FAULT : QOW1 : Charge Outside Window Detected', [251].TIME.YEAR := 2016, [251].TIME.MONTH := 7, [251].TIME.DAY := 16, [251].TIME.HOUR := 9, [251].TIME.MINUTE := 47, [251].TIME.SECOND := 26, [251].TIME.MICROSECOND := 499503, [251].EVENT := '2016/07/16   09:47:26   USER : PPS RESET FAULT BUTTON PRESSED', [252].TIME.YEAR := 2016, [252].TIME.MONTH := 7, [252].TIME.DAY := 16, [252].TIME.HOUR := 9, [252].TIME.MINUTE := 50, [252].TIME.SECOND := 41, [252].TIME.MICROSECOND := 399504, [252].EVENT := '2016/07/16   09:50:41   USER : PPS RESET FAULT BUTTON PRESSED', [253].TIME.YEAR := 2016, [253].TIME.MONTH := 7, [253].TIME.DAY := 16, [253].TIME.HOUR := 13, [253].TIME.MINUTE := 44, [253].TIME.SECOND := 38, [253].TIME.MICROSECOND := 299509, [253].EVENT := '2016/07/16   13:44:38   USER : PPS RESET FAULT BUTTON PRESSED', [254].TIME.YEAR := 2016, [254].TIME.MONTH := 7, [254].TIME.DAY := 18, [254].TIME.HOUR := 15, [254].TIME.MINUTE := 40, [254].TIME.SECOND := 5, [254].TIME.MICROSECOND := 300019, [254].EVENT := '2016/07/18   15:40:05   USER : PPS RESET FAULT BUTTON PRESSED', [255].TIME.YEAR := 2016, [255].TIME.MONTH := 7, [255].TIME.DAY := 18, [255].TIME.HOUR := 16, [255].TIME.MINUTE := 23, [255].TIME.SECOND := 20, [255].TIME.MICROSECOND := 599515, [255].EVENT := '2016/07/18   16:23:20   FAULT : QOW1 : Charge Outside Window Detected', [256].TIME.YEAR := 2016, [256].TIME.MONTH := 7, [256].TIME.DAY := 18, [256].TIME.HOUR := 16, [256].TIME.MINUTE := 23, [256].TIME.SECOND := 49,
        [256].TIME.MICROSECOND := 199510, [256].EVENT := '2016/07/18   16:23:49   USER : PPS RESET FAULT BUTTON PRESSED', [257].TIME.YEAR := 2016, [257].TIME.MONTH := 7, [257].TIME.DAY := 19, [257].TIME.HOUR := 12, [257].TIME.MINUTE := 12, [257].TIME.SECOND := 54, [257].TIME.MICROSECOND := 899507, [257].EVENT := '2016/07/19   12:12:54   USER : PPS RESET FAULT BUTTON PRESSED', [258].TIME.YEAR := 2016, [258].TIME.MONTH := 7, [258].TIME.DAY := 20, [258].TIME.MINUTE := 8, [258].TIME.SECOND := 41, [258].TIME.MICROSECOND := 599943, [258].EVENT := '2016/07/20   00:08:41   USER : PPS RESET FAULT BUTTON PRESSED', [259].TIME.YEAR := 2016, [259].TIME.MONTH := 7, [259].TIME.DAY := 20, [259].TIME.MINUTE := 8, [259].TIME.SECOND := 50, [259].TIME.MICROSECOND := 599513, [259].EVENT := '2016/07/20   00:08:50   USER : PPS RESET FAULT BUTTON PRESSED', [260].TIME.YEAR := 2016, [260].TIME.MONTH := 7, [260].TIME.DAY := 20, [260].TIME.HOUR := 9, [260].TIME.MINUTE := 17, [260].TIME.SECOND := 19, [260].TIME.MICROSECOND := 500111, [260].EVENT := '2016/07/20   09:17:19   FAULT : QOW1 : Charge Outside Window Detected', [261].TIME.YEAR := 2016, [261].TIME.MONTH := 7, [261].TIME.DAY := 20, [261].TIME.HOUR := 9, [261].TIME.MINUTE := 17, [261].TIME.SECOND := 19, [261].TIME.MICROSECOND := 699514, [261].EVENT := '2016/07/20   09:17:19   USER : PPS RESET FAULT BUTTON PRESSED', [262].TIME.YEAR := 2016, [262].TIME.MONTH := 7, [262].TIME.DAY := 20, [262].TIME.HOUR := 9, [262].TIME.MINUTE := 17, [262].TIME.SECOND := 23, [262].TIME.MICROSECOND := 899507, [262].EVENT := '2016/07/20   09:17:23   USER : PPS RESET FAULT BUTTON PRESSED', [263].TIME.YEAR := 2016, [263].TIME.MONTH := 7, [263].TIME.DAY := 20, [263].TIME.HOUR := 9, [263].TIME.MINUTE := 39, [263].TIME.SECOND := 57, [263].TIME.MICROSECOND := 699503, [263].EVENT := '2016/07/20   09:39:57   USER : PPS RESET FAULT BUTTON PRESSED', [264].TIME.YEAR := 2016, [264].TIME.MONTH := 7, [264].TIME.DAY := 20, [264].TIME.HOUR := 9,
        [264].TIME.MINUTE := 43, [264].TIME.SECOND := 13, [264].TIME.MICROSECOND := 800024, [264].EVENT := '2016/07/20   09:43:13   USER : PPS RESET FAULT BUTTON PRESSED', [265].TIME.YEAR := 2016, [265].TIME.MONTH := 7, [265].TIME.DAY := 20, [265].TIME.HOUR := 9, [265].TIME.MINUTE := 43, [265].TIME.SECOND := 18, [265].TIME.MICROSECOND := 899941, [265].EVENT := '2016/07/20   09:43:18   USER : PPS RESET FAULT BUTTON PRESSED', [266].TIME.YEAR := 2016, [266].TIME.MONTH := 7, [266].TIME.DAY := 20, [266].TIME.HOUR := 9, [266].TIME.MINUTE := 50, [266].TIME.SECOND := 46, [266].TIME.MICROSECOND := 299518, [266].EVENT := '2016/07/20   09:50:46   USER : PPS RESET FAULT BUTTON PRESSED', [267].TIME.YEAR := 2016, [267].TIME.MONTH := 7, [267].TIME.DAY := 20, [267].TIME.HOUR := 9, [267].TIME.MINUTE := 50, [267].TIME.SECOND := 50, [267].TIME.MICROSECOND := 200021, [267].EVENT := '2016/07/20   09:50:50   USER : PPS RESET FAULT BUTTON PRESSED', [268].TIME.YEAR := 2016, [268].TIME.MONTH := 7, [268].TIME.DAY := 20, [268].TIME.HOUR := 10, [268].TIME.MINUTE := 8, [268].TIME.SECOND := 50, [268].TIME.MICROSECOND := 999510, [268].EVENT := '2016/07/20   10:08:50   USER : PPS RESET FAULT BUTTON PRESSED', [269].TIME.YEAR := 2016, [269].TIME.MONTH := 7, [269].TIME.DAY := 20, [269].TIME.HOUR := 10, [269].TIME.MINUTE := 8, [269].TIME.SECOND := 53, [269].TIME.MICROSECOND := 599506, [269].EVENT := '2016/07/20   10:08:53   USER : PPS RESET FAULT BUTTON PRESSED', [270].TIME.YEAR := 2016, [270].TIME.MONTH := 7, [270].TIME.DAY := 20, [270].TIME.HOUR := 10, [270].TIME.MINUTE := 8, [270].TIME.SECOND := 56, [270].TIME.MICROSECOND := 499512, [270].EVENT := '2016/07/20   10:08:56   USER : PPS RESET FAULT BUTTON PRESSED', [271].TIME.YEAR := 2016, [271].TIME.MONTH := 7, [271].TIME.DAY := 22, [271].TIME.HOUR := 1, [271].TIME.MINUTE := 33, [271].TIME.SECOND := 10, [271].TIME.MICROSECOND := 799507, [271].EVENT := '2016/07/22   01:33:10   USER : PPS RESET FAULT BUTTON PRESSED',
        [272].TIME.YEAR := 2016, [272].TIME.MONTH := 7, [272].TIME.DAY := 22, [272].TIME.HOUR := 3, [272].TIME.MINUTE := 28, [272].TIME.SECOND := 28, [272].TIME.MICROSECOND := 800024, [272].EVENT := '2016/07/22   03:28:28   USER : PPS RESET FAULT BUTTON PRESSED', [273].TIME.YEAR := 2016, [273].TIME.MONTH := 7, [273].TIME.DAY := 22, [273].TIME.HOUR := 4, [273].TIME.MINUTE := 9, [273].TIME.SECOND := 23, [273].TIME.MICROSECOND := 799942, [273].EVENT := '2016/07/22   04:09:23   USER : PPS RESET FAULT BUTTON PRESSED', [274].TIME.YEAR := 2016, [274].TIME.MONTH := 7, [274].TIME.DAY := 22, [274].TIME.HOUR := 5, [274].TIME.MINUTE := 15, [274].TIME.SECOND := 46, [274].TIME.MICROSECOND := 499517, [274].EVENT := '2016/07/22   05:15:46   USER : PPS RESET FAULT BUTTON PRESSED', [275].TIME.YEAR := 2016, [275].TIME.MONTH := 7, [275].TIME.DAY := 22, [275].TIME.HOUR := 5, [275].TIME.MINUTE := 15, [275].TIME.SECOND := 51, [275].TIME.MICROSECOND := 499503, [275].EVENT := '2016/07/22   05:15:51   USER : PPS RESET FAULT BUTTON PRESSED', [276].TIME.YEAR := 2016, [276].TIME.MONTH := 7, [276].TIME.DAY := 22, [276].TIME.HOUR := 5, [276].TIME.MINUTE := 16, [276].TIME.SECOND := 54, [276].TIME.MICROSECOND := 899945, [276].EVENT := '2016/07/22   05:16:54   USER : PPS RESET FAULT BUTTON PRESSED', [277].TIME.YEAR := 2016, [277].TIME.MONTH := 7, [277].TIME.DAY := 23, [277].TIME.HOUR := 7, [277].TIME.MINUTE := 46, [277].TIME.SECOND := 38, [277].TIME.MICROSECOND := 699506, [277].EVENT := '2016/07/23   07:46:38   USER : PPS RESET FAULT BUTTON PRESSED', [278].TIME.YEAR := 2016, [278].TIME.MONTH := 7, [278].TIME.DAY := 23, [278].TIME.HOUR := 7, [278].TIME.MINUTE := 46, [278].TIME.SECOND := 41, [278].TIME.MICROSECOND := 799509, [278].EVENT := '2016/07/23   07:46:41   USER : PPS RESET FAULT BUTTON PRESSED', [279].TIME.YEAR := 2016, [279].TIME.MONTH := 7, [279].TIME.DAY := 23, [279].TIME.HOUR := 12,
        [279].TIME.MINUTE := 33, [279].TIME.SECOND := 12, [279].TIME.MICROSECOND := 199939, [279].EVENT := '2016/07/23   12:33:12   USER : PPS RESET FAULT BUTTON PRESSED', [280].TIME.YEAR := 2016, [280].TIME.MONTH := 7, [280].TIME.DAY := 24, [280].TIME.HOUR := 4, [280].TIME.MINUTE := 44, [280].TIME.SECOND := 48, [280].TIME.MICROSECOND := 699555, [280].EVENT := '2016/07/24   04:44:48   USER : PPS RESET FAULT BUTTON PRESSED', [281].TIME.YEAR := 2016, [281].TIME.MONTH := 7, [281].TIME.DAY := 24, [281].TIME.HOUR := 4, [281].TIME.MINUTE := 58, [281].TIME.SECOND := 2, [281].TIME.MICROSECOND := 900019, [281].EVENT := '2016/07/24   04:58:02   USER : PPS RESET FAULT BUTTON PRESSED', [282].TIME.YEAR := 2016, [282].TIME.MONTH := 7, [282].TIME.DAY := 24, [282].TIME.HOUR := 8, [282].TIME.MINUTE := 52, [282].TIME.SECOND := 6, [282].TIME.MICROSECOND := 999465, [282].EVENT := '2016/07/24   08:52:06   FAULT : QOW1 : Charge Outside Window Detected', [283].TIME.YEAR := 2016, [283].TIME.MONTH := 7, [283].TIME.DAY := 24, [283].TIME.HOUR := 9, [283].TIME.MINUTE := 41, [283].TIME.SECOND := 40, [283].TIME.MICROSECOND := 199510, [283].EVENT := '2016/07/24   09:41:40   USER : PPS RESET FAULT BUTTON PRESSED', [284].TIME.YEAR := 2016, [284].TIME.MONTH := 7, [284].TIME.DAY := 24, [284].TIME.HOUR := 16, [284].TIME.MINUTE := 8, [284].TIME.SECOND := 54, [284].TIME.MICROSECOND := 199939, [284].EVENT := '2016/07/24   16:08:54   USER : PPS RESET FAULT BUTTON PRESSED', [285].TIME.YEAR := 2016, [285].TIME.MONTH := 7, [285].TIME.DAY := 24, [285].TIME.HOUR := 16, [285].TIME.MINUTE := 20, [285].TIME.SECOND := 21, [285].TIME.MICROSECOND := 299463, [285].EVENT := '2016/07/24   16:20:21   FAULT : QOW1 : Charge Outside Window Detected', [286].TIME.YEAR := 2016, [286].TIME.MONTH := 7, [286].TIME.DAY := 24, [286].TIME.HOUR := 16, [286].TIME.MINUTE := 21, [286].TIME.SECOND := 27, [286].TIME.MICROSECOND := 699946, [286].EVENT := '2016/07/24   16:21:27   USER : PPS RESET FAULT BUTTON PRESSED',
        [287].TIME.YEAR := 2016, [287].TIME.MONTH := 7, [287].TIME.DAY := 24, [287].TIME.HOUR := 16, [287].TIME.MINUTE := 21, [287].TIME.SECOND := 33, [287].TIME.MICROSECOND := 399506, [287].EVENT := '2016/07/24   16:21:33   USER : PPS RESET FAULT BUTTON PRESSED', [288].TIME.YEAR := 2016, [288].TIME.MONTH := 7, [288].TIME.DAY := 25, [288].TIME.HOUR := 9, [288].TIME.MINUTE := 17, [288].TIME.SECOND := 44, [288].TIME.MICROSECOND := 499622, [288].EVENT := '2016/07/25   09:17:44   USER : PPS RESET FAULT BUTTON PRESSED', [289].TIME.YEAR := 2016, [289].TIME.MONTH := 7, [289].TIME.DAY := 25, [289].TIME.HOUR := 12, [289].TIME.MINUTE := 24, [289].TIME.SECOND := 21, [289].TIME.MICROSECOND := 499508, [289].EVENT := '2016/07/25   12:24:21   USER : PPS RESET FAULT BUTTON PRESSED', [290].TIME.YEAR := 2016, [290].TIME.MONTH := 7, [290].TIME.DAY := 25, [290].TIME.HOUR := 12, [290].TIME.MINUTE := 47, [290].TIME.SECOND := 30, [290].TIME.MICROSECOND := 799460, [290].EVENT := '2016/07/25   12:47:30   FAULT : QOW1 : Charge Outside Window Detected', [291].TIME.YEAR := 2016, [291].TIME.MONTH := 7, [291].TIME.DAY := 25, [291].TIME.HOUR := 15, [291].TIME.MINUTE := 59, [291].TIME.SECOND := 51, [291].TIME.MICROSECOND := 599932, [291].EVENT := '2016/07/25   15:59:51   USER : PPS RESET FAULT BUTTON PRESSED', [292].TIME.YEAR := 2016, [292].TIME.MONTH := 7, [292].TIME.DAY := 25, [292].TIME.HOUR := 17, [292].TIME.MINUTE := 19, [292].TIME.SECOND := 53, [292].TIME.MICROSECOND := 899510, [292].EVENT := '2016/07/25   17:19:53   USER : PPS RESET FAULT BUTTON PRESSED', [293].TIME.YEAR := 2016, [293].TIME.MONTH := 7, [293].TIME.DAY := 25, [293].TIME.HOUR := 17, [293].TIME.MINUTE := 40, [293].TIME.SECOND := 55, [293].TIME.MICROSECOND := 699548, [293].EVENT := '2016/07/25   17:40:55   USER : PPS RESET FAULT BUTTON PRESSED', [294].TIME.YEAR := 2016, [294].TIME.MONTH := 7, [294].TIME.DAY := 25, [294].TIME.HOUR := 20,
        [294].TIME.MINUTE := 21, [294].TIME.SECOND := 33, [294].TIME.MICROSECOND := 499515, [294].EVENT := '2016/07/25   20:21:33   USER : PPS RESET FAULT BUTTON PRESSED', [295].TIME.YEAR := 2016, [295].TIME.MONTH := 7, [295].TIME.DAY := 25, [295].TIME.HOUR := 20, [295].TIME.MINUTE := 31, [295].TIME.SECOND := 17, [295].TIME.MICROSECOND := 799507, [295].EVENT := '2016/07/25   20:31:17   USER : PPS RESET FAULT BUTTON PRESSED', [296].TIME.YEAR := 2016, [296].TIME.MONTH := 7, [296].TIME.DAY := 25, [296].TIME.HOUR := 22, [296].TIME.MINUTE := 43, [296].TIME.SECOND := 40, [296].TIME.MICROSECOND := 199507, [296].EVENT := '2016/07/25   22:43:40   USER : PPS RESET FAULT BUTTON PRESSED', [297].TIME.YEAR := 2016, [297].TIME.MONTH := 7, [297].TIME.DAY := 26, [297].TIME.HOUR := 9, [297].TIME.MINUTE := 9, [297].TIME.SECOND := 51, [297].TIME.MICROSECOND := 799571, [297].EVENT := '2016/07/26   09:09:51   USER : PPS RESET FAULT BUTTON PRESSED', [298].TIME.YEAR := 2016, [298].TIME.MONTH := 7, [298].TIME.DAY := 26, [298].TIME.HOUR := 9, [298].TIME.MINUTE := 11, [298].TIME.SECOND := 14, [298].TIME.MICROSECOND := 199503, [298].EVENT := '2016/07/26   09:11:14   USER : PPS RESET FAULT BUTTON PRESSED', [299].TIME.YEAR := 2016, [299].TIME.MONTH := 7, [299].TIME.DAY := 26, [299].TIME.HOUR := 9, [299].TIME.MINUTE := 11, [299].TIME.SECOND := 50, [299].TIME.MICROSECOND := 399507, [299].EVENT := '2016/07/26   09:11:50   USER : PPS RESET FAULT BUTTON PRESSED', [300].TIME.YEAR := 2016, [300].TIME.MONTH := 7, [300].TIME.DAY := 26, [300].TIME.HOUR := 9, [300].TIME.MINUTE := 15, [300].TIME.SECOND := 27, [300].TIME.MICROSECOND := 899506, [300].EVENT := '2016/07/26   09:15:27   USER : PPS RESET FAULT BUTTON PRESSED', [301].TIME.YEAR := 2016, [301].TIME.MONTH := 7, [301].TIME.DAY := 26, [301].TIME.HOUR := 9, [301].TIME.MINUTE := 24, [301].TIME.SECOND := 10, [301].TIME.MICROSECOND := 99512, [301].EVENT := '2016/07/26   09:24:10   USER : PPS RESET FAULT BUTTON PRESSED',
        [302].TIME.YEAR := 2016, [302].TIME.MONTH := 7, [302].TIME.DAY := 26, [302].TIME.HOUR := 9, [302].TIME.MINUTE := 32, [302].TIME.SECOND := 4, [302].TIME.MICROSECOND := 799465, [302].EVENT := '2016/07/26   09:32:04   FAULT : QOW1 : Charge Outside Window Detected', [303].TIME.YEAR := 2016, [303].TIME.MONTH := 7, [303].TIME.DAY := 26, [303].TIME.HOUR := 9, [303].TIME.MINUTE := 32, [303].TIME.SECOND := 5, [303].TIME.MICROSECOND := 200023, [303].EVENT := '2016/07/26   09:32:05   USER : PPS RESET FAULT BUTTON PRESSED', [304].TIME.YEAR := 2016, [304].TIME.MONTH := 7, [304].TIME.DAY := 26, [304].TIME.HOUR := 15, [304].TIME.MINUTE := 11, [304].TIME.SECOND := 39, [304].TIME.MICROSECOND := 99511, [304].EVENT := '2016/07/26   15:11:39   USER : PPS RESET FAULT BUTTON PRESSED', [305].TIME.YEAR := 2016, [305].TIME.MONTH := 7, [305].TIME.DAY := 26, [305].TIME.HOUR := 20, [305].TIME.MINUTE := 20, [305].TIME.SECOND := 51, [305].TIME.MICROSECOND := 799509, [305].EVENT := '2016/07/26   20:20:51   USER : PPS RESET FAULT BUTTON PRESSED', [306].TIME.YEAR := 2016, [306].TIME.MONTH := 7, [306].TIME.DAY := 26, [306].TIME.HOUR := 20, [306].TIME.MINUTE := 20, [306].TIME.SECOND := 52, [306].TIME.MICROSECOND := 399508, [306].EVENT := '2016/07/26   20:20:52   USER : PPS RESET FAULT BUTTON PRESSED', [307].TIME.YEAR := 2016, [307].TIME.MONTH := 7, [307].TIME.DAY := 26, [307].TIME.HOUR := 20, [307].TIME.MINUTE := 20, [307].TIME.SECOND := 52, [307].TIME.MICROSECOND := 599505, [307].EVENT := '2016/07/26   20:20:52   USER : PPS RESET FAULT BUTTON PRESSED', [308].TIME.YEAR := 2016, [308].TIME.MONTH := 7, [308].TIME.DAY := 26, [308].TIME.HOUR := 20, [308].TIME.MINUTE := 20, [308].TIME.SECOND := 52, [308].TIME.MICROSECOND := 899506, [308].EVENT := '2016/07/26   20:20:52   USER : PPS RESET FAULT BUTTON PRESSED', [309].TIME.YEAR := 2016, [309].TIME.MONTH := 7, [309].TIME.DAY := 27, [309].TIME.HOUR := 9,
        [309].TIME.MINUTE := 5, [309].TIME.SECOND := 12, [309].TIME.MICROSECOND := 299938, [309].EVENT := '2016/07/27   09:05:12   USER : PPS RESET FAULT BUTTON PRESSED', [310].TIME.YEAR := 2016, [310].TIME.MONTH := 7, [310].TIME.DAY := 27, [310].TIME.HOUR := 12, [310].TIME.MINUTE := 56, [310].TIME.SECOND := 58, [310].TIME.MICROSECOND := 599941, [310].EVENT := '2016/07/27   12:56:58   USER : PPS RESET FAULT BUTTON PRESSED', [311].TIME.YEAR := 2016, [311].TIME.MONTH := 7, [311].TIME.DAY := 27, [311].TIME.HOUR := 12, [311].TIME.MINUTE := 57, [311].TIME.SECOND := 4, [311].TIME.MICROSECOND := 899652, [311].EVENT := '2016/07/27   12:57:04   USER : PPS RESET FAULT BUTTON PRESSED', [312].TIME.YEAR := 2016, [312].TIME.MONTH := 7, [312].TIME.DAY := 27, [312].TIME.HOUR := 15, [312].TIME.MINUTE := 29, [312].TIME.SECOND := 17, [312].TIME.MICROSECOND := 299508, [312].EVENT := '2016/07/27   15:29:17   USER : PPS RESET FAULT BUTTON PRESSED', [313].TIME.YEAR := 2016, [313].TIME.MONTH := 7, [313].TIME.DAY := 27, [313].TIME.HOUR := 16, [313].TIME.MINUTE := 48, [313].TIME.SECOND := 9, [313].TIME.MICROSECOND := 499509, [313].EVENT := '2016/07/27   16:48:09   USER : PPS RESET FAULT BUTTON PRESSED', [314].TIME.YEAR := 2016, [314].TIME.MONTH := 7, [314].TIME.DAY := 27, [314].TIME.HOUR := 17, [314].TIME.MINUTE := 8, [314].TIME.SECOND := 43, [314].TIME.MICROSECOND := 599508, [314].EVENT := '2016/07/27   17:08:43   USER : PPS RESET FAULT BUTTON PRESSED', [315].TIME.YEAR := 2016, [315].TIME.MONTH := 7, [315].TIME.DAY := 27, [315].TIME.HOUR := 17, [315].TIME.MINUTE := 9, [315].TIME.SECOND := 50, [315].TIME.MICROSECOND := 199511, [315].EVENT := '2016/07/27   17:09:50   USER : PPS RESET FAULT BUTTON PRESSED', [316].TIME.YEAR := 2016, [316].TIME.MONTH := 7, [316].TIME.DAY := 27, [316].TIME.HOUR := 17, [316].TIME.MINUTE := 25, [316].TIME.SECOND := 11, [316].TIME.MICROSECOND := 499984, [316].EVENT := '2016/07/27   17:25:11   FAULT : QOW1 : Charge Outside Window Detected',
        [317].TIME.YEAR := 2016, [317].TIME.MONTH := 7, [317].TIME.DAY := 27, [317].TIME.HOUR := 17, [317].TIME.MINUTE := 40, [317].TIME.SECOND := 40, [317].TIME.MICROSECOND := 99544, [317].EVENT := '2016/07/27   17:40:40   USER : PPS RESET FAULT BUTTON PRESSED', [318].TIME.YEAR := 2016, [318].TIME.MONTH := 7, [318].TIME.DAY := 27, [318].TIME.HOUR := 17, [318].TIME.MINUTE := 40, [318].TIME.SECOND := 54, [318].TIME.MICROSECOND := 799514, [318].EVENT := '2016/07/27   17:40:54   USER : PPS RESET FAULT BUTTON PRESSED', [319].TIME.YEAR := 2016, [319].TIME.MONTH := 7, [319].TIME.DAY := 27, [319].TIME.HOUR := 18, [319].TIME.MINUTE := 32, [319].TIME.SECOND := 36, [319].TIME.MICROSECOND := 999457, [319].EVENT := '2016/07/27   18:32:36   FAULT : WDT : Trigger Rate LOW', [320].TIME.YEAR := 2016, [320].TIME.MONTH := 7, [320].TIME.DAY := 27, [320].TIME.HOUR := 18, [320].TIME.MINUTE := 32, [320].TIME.SECOND := 59, [320].TIME.MICROSECOND := 499511, [320].EVENT := '2016/07/27   18:32:59   USER : PPS RESET FAULT BUTTON PRESSED', [321].TIME.YEAR := 2016, [321].TIME.MONTH := 7, [321].TIME.DAY := 27, [321].TIME.HOUR := 18, [321].TIME.MINUTE := 42, [321].TIME.SECOND := 54, [321].TIME.MICROSECOND := 499468, [321].EVENT := '2016/07/27   18:42:54   FAULT : WDT : Trigger Rate LOW', [322].TIME.YEAR := 2016, [322].TIME.MONTH := 7, [322].TIME.DAY := 27, [322].TIME.HOUR := 18, [322].TIME.MINUTE := 42, [322].TIME.SECOND := 54, [322].TIME.MICROSECOND := 599463, [322].EVENT := '2016/07/27   18:42:54   FAULT : QOW1 : Charge Outside Window Detected', [323].TIME.YEAR := 2016, [323].TIME.MONTH := 7, [323].TIME.DAY := 27, [323].TIME.HOUR := 18, [323].TIME.MINUTE := 43, [323].TIME.SECOND := 18, [323].TIME.MICROSECOND := 900272, [323].EVENT := '2016/07/27   18:43:18   USER : PPS RESET FAULT BUTTON PRESSED', [324].TIME.YEAR := 2016, [324].TIME.MONTH := 7, [324].TIME.DAY := 27, [324].TIME.HOUR := 19,
        [324].TIME.MINUTE := 39, [324].TIME.SECOND := 54, [324].TIME.MICROSECOND := 99578, [324].EVENT := '2016/07/27   19:39:54   USER : PPS RESET FAULT BUTTON PRESSED', [325].TIME.YEAR := 2016, [325].TIME.MONTH := 7, [325].TIME.DAY := 27, [325].TIME.HOUR := 19, [325].TIME.MINUTE := 55, [325].TIME.SECOND := 11, [325].TIME.MICROSECOND := 400021, [325].EVENT := '2016/07/27   19:55:11   USER : PPS RESET FAULT BUTTON PRESSED', [326].TIME.YEAR := 2016, [326].TIME.MONTH := 7, [326].TIME.DAY := 27, [326].TIME.HOUR := 19, [326].TIME.MINUTE := 55, [326].TIME.SECOND := 11, [326].TIME.MICROSECOND := 999516, [326].EVENT := '2016/07/27   19:55:11   USER : PPS RESET FAULT BUTTON PRESSED', [327].TIME.YEAR := 2016, [327].TIME.MONTH := 7, [327].TIME.DAY := 28, [327].TIME.HOUR := 6, [327].TIME.MINUTE := 30, [327].TIME.SECOND := 12, [327].TIME.MICROSECOND := 899510, [327].EVENT := '2016/07/28   06:30:12   USER : PPS RESET FAULT BUTTON PRESSED', [328].TIME.YEAR := 2016, [328].TIME.MONTH := 7, [328].TIME.DAY := 29, [328].TIME.HOUR := 20, [328].TIME.MINUTE := 57, [328].TIME.SECOND := 51, [328].TIME.MICROSECOND := 599506, [328].EVENT := '2016/07/29   20:57:51   USER : PPS RESET FAULT BUTTON PRESSED', [329].TIME.YEAR := 2016, [329].TIME.MONTH := 7, [329].TIME.DAY := 29, [329].TIME.HOUR := 20, [329].TIME.MINUTE := 57, [329].TIME.SECOND := 57, [329].TIME.MICROSECOND := 600087, [329].EVENT := '2016/07/29   20:57:57   USER : PPS RESET FAULT BUTTON PRESSED', [330].TIME.YEAR := 2016, [330].TIME.MONTH := 7, [330].TIME.DAY := 29, [330].TIME.HOUR := 20, [330].TIME.MINUTE := 58, [330].TIME.SECOND := 1, [330].TIME.MICROSECOND := 999508, [330].EVENT := '2016/07/29   20:58:01   USER : PPS RESET FAULT BUTTON PRESSED', [331].TIME.YEAR := 2016, [331].TIME.MONTH := 7, [331].TIME.DAY := 30, [331].TIME.MINUTE := 44, [331].TIME.SECOND := 52, [331].TIME.MICROSECOND := 899515, [331].EVENT := '2016/07/30   00:44:52   USER : PPS RESET FAULT BUTTON PRESSED', [332].TIME.YEAR := 2016,
        [332].TIME.MONTH := 7, [332].TIME.DAY := 30, [332].TIME.MINUTE := 44, [332].TIME.SECOND := 58, [332].TIME.MICROSECOND := 99510, [332].EVENT := '2016/07/30   00:44:58   USER : PPS RESET FAULT BUTTON PRESSED', [333].TIME.YEAR := 2016, [333].TIME.MONTH := 7, [333].TIME.DAY := 30, [333].TIME.HOUR := 1, [333].TIME.MINUTE := 2, [333].TIME.SECOND := 29, [333].TIME.MICROSECOND := 499653, [333].EVENT := '2016/07/30   01:02:29   USER : PPS RESET FAULT BUTTON PRESSED', [334].TIME.YEAR := 2016, [334].TIME.MONTH := 7, [334].TIME.DAY := 30, [334].TIME.HOUR := 1, [334].TIME.MINUTE := 49, [334].TIME.SECOND := 37, [334].TIME.MICROSECOND := 999562, [334].EVENT := '2016/07/30   01:49:37   USER : PPS RESET FAULT BUTTON PRESSED', [335].TIME.YEAR := 2016, [335].TIME.MONTH := 7, [335].TIME.DAY := 31, [335].TIME.HOUR := 20, [335].TIME.MINUTE := 36, [335].TIME.SECOND := 43, [335].TIME.MICROSECOND := 199513, [335].EVENT := '2016/07/31   20:36:43   USER : PPS RESET FAULT BUTTON PRESSED', [336].TIME.YEAR := 2016, [336].TIME.MONTH := 7, [336].TIME.DAY := 31, [336].TIME.HOUR := 20, [336].TIME.MINUTE := 38, [336].TIME.SECOND := 23, [336].TIME.MICROSECOND := 399511, [336].EVENT := '2016/07/31   20:38:23   USER : PPS RESET FAULT BUTTON PRESSED', [337].TIME.YEAR := 2016, [337].TIME.MONTH := 8, [337].TIME.DAY := 2, [337].TIME.HOUR := 5, [337].TIME.MINUTE := 34, [337].TIME.SECOND := 16, [337].TIME.MICROSECOND := 699463, [337].EVENT := '2016/08/02   05:34:16   FAULT : QOW1 : Charge Outside Window Detected', [338].TIME.YEAR := 2016, [338].TIME.MONTH := 8, [338].TIME.DAY := 2, [338].TIME.HOUR := 5, [338].TIME.MINUTE := 37, [338].TIME.SECOND := 29, [338].TIME.MICROSECOND := 399507, [338].EVENT := '2016/08/02   05:37:29   USER : PPS RESET FAULT BUTTON PRESSED', [339].TIME.YEAR := 2016, [339].TIME.MONTH := 8, [339].TIME.DAY := 2, [339].TIME.HOUR := 9, [339].TIME.MINUTE := 6, [339].TIME.SECOND := 42,
        [339].TIME.MICROSECOND := 999511, [339].EVENT := '2016/08/02   09:06:42   USER : PPS RESET FAULT BUTTON PRESSED', [340].TIME.YEAR := 2016, [340].TIME.MONTH := 8, [340].TIME.DAY := 2, [340].TIME.HOUR := 22, [340].TIME.MINUTE := 24, [340].TIME.SECOND := 15, [340].TIME.MICROSECOND := 199461, [340].EVENT := '2016/08/02   22:24:15   FAULT : QOW1 : Charge Outside Window Detected', [341].TIME.YEAR := 2016, [341].TIME.MONTH := 8, [341].TIME.DAY := 2, [341].TIME.HOUR := 22, [341].TIME.MINUTE := 29, [341].TIME.SECOND := 58, [341].TIME.MICROSECOND := 99515, [341].EVENT := '2016/08/02   22:29:58   USER : PPS RESET FAULT BUTTON PRESSED', [342].TIME.YEAR := 2016, [342].TIME.MONTH := 8, [342].TIME.DAY := 4, [342].TIME.HOUR := 13, [342].TIME.MINUTE := 34, [342].TIME.SECOND := 47, [342].TIME.MICROSECOND := 99458, [342].EVENT := '2016/08/04   13:34:47   FAULT : QOW1 : Charge Outside Window Detected', [343].TIME.YEAR := 2016, [343].TIME.MONTH := 8, [343].TIME.DAY := 4, [343].TIME.HOUR := 13, [343].TIME.MINUTE := 45, [343].TIME.SECOND := 23, [343].TIME.MICROSECOND := 999509, [343].EVENT := '2016/08/04   13:45:23   USER : PPS RESET FAULT BUTTON PRESSED', [344].TIME.YEAR := 2016, [344].TIME.MONTH := 8, [344].TIME.DAY := 5, [344].TIME.HOUR := 10, [344].TIME.MINUTE := 7, [344].TIME.SECOND := 10, [344].TIME.MICROSECOND := 599464, [344].EVENT := '2016/08/05   10:07:10   FAULT : QOW1 : Charge Outside Window Detected', [345].TIME.YEAR := 2016, [345].TIME.MONTH := 8, [345].TIME.DAY := 5, [345].TIME.HOUR := 10, [345].TIME.MINUTE := 11, [345].TIME.SECOND := 45, [345].TIME.MICROSECOND := 799513, [345].EVENT := '2016/08/05   10:11:45   USER : PPS RESET FAULT BUTTON PRESSED', [346].TIME.YEAR := 2016, [346].TIME.MONTH := 8, [346].TIME.DAY := 5, [346].TIME.HOUR := 10, [346].TIME.MINUTE := 13, [346].TIME.SECOND := 34, [346].TIME.MICROSECOND := 299501, [346].EVENT := '2016/08/05   10:13:34   USER : PPS RESET FAULT BUTTON PRESSED', [347].TIME.YEAR := 2016, [347].TIME.MONTH := 8,
        [347].TIME.DAY := 5, [347].TIME.HOUR := 10, [347].TIME.MINUTE := 35, [347].TIME.SECOND := 1, [347].TIME.MICROSECOND := 599609, [347].EVENT := '2016/08/05   10:35:01   USER : PPS RESET FAULT BUTTON PRESSED', [348].TIME.YEAR := 2016, [348].TIME.MONTH := 8, [348].TIME.DAY := 5, [348].TIME.HOUR := 10, [348].TIME.MINUTE := 49, [348].TIME.SECOND := 51, [348].TIME.MICROSECOND := 199509, [348].EVENT := '2016/08/05   10:49:51   USER : PPS RESET FAULT BUTTON PRESSED', [349].TIME.YEAR := 2016, [349].TIME.MONTH := 8, [349].TIME.DAY := 5, [349].TIME.HOUR := 10, [349].TIME.MINUTE := 49, [349].TIME.SECOND := 53, [349].TIME.MICROSECOND := 499512, [349].EVENT := '2016/08/05   10:49:53   USER : PPS RESET FAULT BUTTON PRESSED', [350].TIME.YEAR := 2016, [350].TIME.MONTH := 8, [350].TIME.DAY := 5, [350].TIME.HOUR := 10, [350].TIME.MINUTE := 49, [350].TIME.SECOND := 58, [350].TIME.MICROSECOND := 599510, [350].EVENT := '2016/08/05   10:49:58   USER : PPS RESET FAULT BUTTON PRESSED', [351].TIME.YEAR := 2016, [351].TIME.MONTH := 8, [351].TIME.DAY := 5, [351].TIME.HOUR := 11, [351].TIME.MINUTE := 1, [351].TIME.SECOND := 22, [351].TIME.MICROSECOND := 999506, [351].EVENT := '2016/08/05   11:01:22   USER : PPS RESET FAULT BUTTON PRESSED', [352].TIME.YEAR := 2016, [352].TIME.MONTH := 8, [352].TIME.DAY := 5, [352].TIME.HOUR := 11, [352].TIME.MINUTE := 2, [352].TIME.SECOND := 17, [352].TIME.MICROSECOND := 99505, [352].EVENT := '2016/08/05   11:02:17   USER : PPS RESET FAULT BUTTON PRESSED', [353].TIME.YEAR := 2016, [353].TIME.MONTH := 8, [353].TIME.DAY := 5, [353].TIME.HOUR := 14, [353].TIME.MINUTE := 41, [353].TIME.SECOND := 35, [353].TIME.MICROSECOND := 99941, [353].EVENT := '2016/08/05   14:41:35   USER : PPS RESET FAULT BUTTON PRESSED', [354].TIME.YEAR := 2016, [354].TIME.MONTH := 8, [354].TIME.DAY := 5, [354].TIME.HOUR := 14, [354].TIME.MINUTE := 42, [354].TIME.SECOND := 14,
        [354].TIME.MICROSECOND := 199510, [354].EVENT := '2016/08/05   14:42:14   USER : PPS RESET FAULT BUTTON PRESSED', [355].TIME.YEAR := 2016, [355].TIME.MONTH := 8, [355].TIME.DAY := 6, [355].TIME.HOUR := 6, [355].TIME.MINUTE := 22, [355].TIME.SECOND := 32, [355].TIME.MICROSECOND := 899982, [355].EVENT := '2016/08/06   06:22:32   FAULT : QOW1 : Charge Outside Window Detected', [356].TIME.YEAR := 2016, [356].TIME.MONTH := 8, [356].TIME.DAY := 6, [356].TIME.HOUR := 6, [356].TIME.MINUTE := 31, [356].TIME.SECOND := 4, [356].TIME.MICROSECOND := 900021, [356].EVENT := '2016/08/06   06:31:04   USER : PPS RESET FAULT BUTTON PRESSED', [357].TIME.YEAR := 2016, [357].TIME.MONTH := 8, [357].TIME.DAY := 6, [357].TIME.HOUR := 6, [357].TIME.MINUTE := 54, [357].TIME.SECOND := 57, [357].TIME.MICROSECOND := 35, [357].EVENT := '2016/08/06   06:54:57   USER : PPS RESET FAULT BUTTON PRESSED', [358].TIME.YEAR := 2016, [358].TIME.MONTH := 8, [358].TIME.DAY := 6, [358].TIME.HOUR := 7, [358].TIME.MINUTE := 10, [358].TIME.SECOND := 11, [358].TIME.MICROSECOND := 199462, [358].EVENT := '2016/08/06   07:10:11   FAULT : QOW1 : Charge Outside Window Detected', [359].TIME.YEAR := 2016, [359].TIME.MONTH := 8, [359].TIME.DAY := 6, [359].TIME.HOUR := 7, [359].TIME.MINUTE := 10, [359].TIME.SECOND := 19, [359].TIME.MICROSECOND := 999711, [359].EVENT := '2016/08/06   07:10:19   USER : PPS RESET FAULT BUTTON PRESSED', [360].TIME.YEAR := 2016, [360].TIME.MONTH := 8, [360].TIME.DAY := 6, [360].TIME.HOUR := 7, [360].TIME.MINUTE := 16, [360].TIME.SECOND := 2, [360].TIME.MICROSECOND := 599504, [360].EVENT := '2016/08/06   07:16:02   USER : PPS RESET FAULT BUTTON PRESSED', [361].TIME.YEAR := 2016, [361].TIME.MONTH := 8, [361].TIME.DAY := 6, [361].TIME.HOUR := 9, [361].TIME.MINUTE := 35, [361].TIME.SECOND := 34, [361].TIME.MICROSECOND := 99508, [361].EVENT := '2016/08/06   09:35:34   USER : PPS RESET FAULT BUTTON PRESSED', [362].TIME.YEAR := 2016, [362].TIME.MONTH := 8,
